LIN {X 0,Y 474.185,Z 288.904,A -85,B 0,C 180,E1 -7449.626,E2 -7449.626} C_VEL
LIN {X 0,Y 468.545,Z 295.09,A -85,B 0,C 180,E1 -7449.509,E2 -7449.509} C_VEL
LIN {X 0,Y 466.901,Z 298.538,A -85,B 0,C 180,E1 -7449.489,E2 -7449.489} C_VEL
LIN {X 0,Y 466.86,Z 301.446,A -85,B 0,C 180,E1 -7449.52,E2 -7449.52} C_VEL
LIN {X 0,Y 468.004,Z 304.741,A -85,B 0,C 180,E1 -7449.617,E2 -7449.617} C_VEL
LIN {X 0,Y 472.692,Z 312.938,A -85,B 0,C 180,E1 -7449.976,E2 -7449.976} C_VEL
LIN {X 0,Y 473.425,Z 316.419,A -85,B 0,C 180,E1 -7450.068,E2 -7450.068} C_VEL
LIN {X 0,Y 472.347,Z 423.939,A -85,B 0,C 180,E1 -7451.737,E2 -7451.737} C_VEL
LIN {X 0,Y 471.944,Z 437.997,A -85,B 0,C 180,E1 -7452.116,E2 -7452.116} C_VEL
LIN {X 0,Y 471.535,Z 451.556,A -85,B 0,C 180,E1 -7452.657,E2 -7452.657} C_VEL
LIN {X 0,Y 470.962,Z 463.993,A -85,B 0,C 180,E1 -7453.311,E2 -7453.311} C_VEL
LIN {X 0,Y 470.322,Z 476.852,A -85,B 0,C 180,E1 -7454.175,E2 -7454.175} C_VEL
LIN {X 0,Y 469.63,Z 488.571,A -85,B 0,C 180,E1 -7455.151,E2 -7455.151} C_VEL
LIN {X 0,Y 468.872,Z 500.266,A -85,B 0,C 180,E1 -7456.345,E2 -7456.345} C_VEL
LIN {X 0,Y 468.289,Z 510.754,A -85,B 0,C 180,E1 -7457.657,E2 -7457.657} C_VEL
LIN {X 0,Y 467.805,Z 519.328,A -85,B 0,C 180,E1 -7458.957,E2 -7458.957} C_VEL
LIN {X 0,Y 467.34,Z 527.589,A -85,B 0,C 180,E1 -7460.478,E2 -7460.478} C_VEL
LIN {X 0,Y 467.082,Z 533.343,A -85,B 0,C 180,E1 -7461.782,E2 -7461.782} C_VEL
LIN {X 0,Y 466.874,Z 539.353,A -85,B 0,C 180,E1 -7463.475,E2 -7463.475} C_VEL
LIN {X 0,Y 466.775,Z 542.98,A -85,B 0,C 180,E1 -7464.817,E2 -7464.817} C_VEL
LIN {X 0,Y 466.692,Z 546.396,A -85,B 0,C 180,E1 -7466.547,E2 -7466.547} C_VEL
LIN {X 0,Y 466.606,Z 548.426,A -85,B 0,C 180,E1 -7468.274,E2 -7468.274} C_VEL
LIN {X 0,Y 466.598,Z 549.126,A -85,B 0,C 180,E1 -7470,E2 -7470} C_VEL
LIN {X 0,Y 466.605,Z 548.504,A -85,B 0,C 180,E1 -7471.726,E2 -7471.726} C_VEL
LIN {X 0,Y 466.692,Z 546.544,A -85,B 0,C 180,E1 -7473.453,E2 -7473.453} C_VEL
LIN {X 0,Y 466.775,Z 543.2,A -85,B 0,C 180,E1 -7475.183,E2 -7475.183} C_VEL
LIN {X 0,Y 466.908,Z 538.376,A -85,B 0,C 180,E1 -7476.916,E2 -7476.916} C_VEL
LIN {X 0,Y 467.143,Z 531.917,A -85,B 0,C 180,E1 -7478.653,E2 -7478.653} C_VEL
LIN {X 0,Y 467.481,Z 524.725,A -85,B 0,C 180,E1 -7480.174,E2 -7480.174} C_VEL
LIN {X 0,Y 468.029,Z 515.83,A -85,B 0,C 180,E1 -7481.696,E2 -7481.696} C_VEL
LIN {X 0,Y 468.534,Z 506.485,A -85,B 0,C 180,E1 -7483.003,E2 -7483.003} C_VEL
LIN {X 0,Y 469.149,Z 496.136,A -85,B 0,C 180,E1 -7484.199,E2 -7484.199} C_VEL
LIN {X 0,Y 469.823,Z 484.715,A -85,B 0,C 180,E1 -7485.286,E2 -7485.286} C_VEL
LIN {X 0,Y 470.575,Z 472.057,A -85,B 0,C 180,E1 -7486.262,E2 -7486.262} C_VEL
LIN {X 0,Y 471.222,Z 458.762,A -85,B 0,C 180,E1 -7487.075,E2 -7487.075} C_VEL
LIN {X 0,Y 471.78,Z 444.827,A -85,B 0,C 180,E1 -7487.724,E2 -7487.724} C_VEL
LIN {X 0,Y 472.174,Z 431.019,A -85,B 0,C 180,E1 -7488.186,E2 -7488.186} C_VEL
LIN {X 0,Y 472.481,Z 416.795,A -85,B 0,C 180,E1 -7488.482,E2 -7488.482} C_VEL
LIN {X 0,Y 473.516,Z 306.855,A -85,B 0,C 180,E1 -7490.171,E2 -7490.171} C_VEL
LIN {X 0,Y 469.764,Z 287.63,A -85,B 0,C 180,E1 -7490.662,E2 -7490.662} C_VEL
LIN {X 0,Y 469.727,Z 286.836,A -85,B 0,C 180,E1 -7490.734,E2 -7490.734} C_VEL
LIN {X 0,Y 470.355,Z 273.557,A -85,B 0,C 180,E1 -7493.092,E2 -7493.092} C_VEL
LIN {X 0,Y 468.135,Z 262.406,A -85,B 0,C 180,E1 -7495.281,E2 -7495.281} C_VEL
LIN {X 0,Y 467.627,Z 259.921,A -85,B 0,C 180,E1 -7495.838,E2 -7495.838} C_VEL
LIN {X 0,Y 467.576,Z 259.854,A -85,B 0,C 180,E1 -7498.749,E2 -7498.749} C_VEL
LIN {X 0,Y 467.582,Z 259.864,A -85,B 0,C 180,E1 -7501.739,E2 -7501.739} C_VEL
LIN {X 0,Y 467.565,Z 259.863,A -85,B 0,C 180,E1 -7504.832,E2 -7504.832} C_VEL
LIN {X 0,Y 467.563,Z 259.863,A -85,B 0,C 180,E1 -7508.044,E2 -7508.044} C_VEL
LIN {X 0,Y 467.579,Z 259.863,A -85,B 0,C 180,E1 -7511.277,E2 -7511.277} C_VEL
LIN {X 0,Y 467.563,Z 259.867,A -85,B 0,C 180,E1 -7513.822,E2 -7513.822} C_VEL
LIN {X 0,Y 467.552,Z 259.865,A -85,B 0,C 180,E1 -7516.255,E2 -7516.255} C_VEL
LIN {X 0,Y 467.579,Z 259.848,A -85,B 0,C 180,E1 -7518.722,E2 -7518.722} C_VEL
LIN {X 0,Y 467.569,Z 259.871,A -85,B 0,C 180,E1 -7521.406,E2 -7521.406} C_VEL
LIN {X 0,Y 467.557,Z 259.863,A -85,B 0,C 180,E1 -7524.26,E2 -7524.26} C_VEL
LIN {X 0,Y 467.576,Z 259.848,A -85,B 0,C 180,E1 -7527.32,E2 -7527.32} C_VEL
LIN {X 0,Y 467.572,Z 259.866,A -85,B 0,C 180,E1 -7530.665,E2 -7530.665} C_VEL
LIN {X 0,Y 467.609,Z 259.858,A -85,B 0,C 180,E1 -7533.199,E2 -7533.199} C_VEL
LIN {X 0,Y 467.585,Z 259.864,A -85,B 0,C 180,E1 -7536.468,E2 -7536.468} C_VEL
LIN {X 0,Y 467.614,Z 259.853,A -85,B 0,C 180,E1 -7539.777,E2 -7539.777} C_VEL
LIN {X 0,Y 467.601,Z 259.863,A -85,B 0,C 180,E1 -7542.506,E2 -7542.506} C_VEL
LIN {X 0,Y 467.598,Z 259.858,A -85,B 0,C 180,E1 -7545.196,E2 -7545.196} C_VEL
LIN {X 0,Y 467.648,Z 259.854,A -85,B 0,C 180,E1 -7547.854,E2 -7547.854} C_VEL
LIN {X 0,Y 467.673,Z 259.845,A -85,B 0,C 180,E1 -7551.357,E2 -7551.357} C_VEL
LIN {X 0,Y 467.738,Z 259.843,A -85,B 0,C 180,E1 -7553.962,E2 -7553.962} C_VEL
LIN {X 0,Y 467.851,Z 259.819,A -85,B 0,C 180,E1 -7557.417,E2 -7557.417} C_VEL
LIN {X 0,Y 467.873,Z 259.826,A -85,B 0,C 180,E1 -7560,E2 -7560} C_VEL
LIN {X 0,Y 467.851,Z 259.828,A -85,B 0,C 180,E1 -7562.583,E2 -7562.583} C_VEL
LIN {X 0,Y 467.735,Z 259.843,A -85,B 0,C 180,E1 -7566.037,E2 -7566.037} C_VEL
LIN {X 0,Y 467.673,Z 259.85,A -85,B 0,C 180,E1 -7568.643,E2 -7568.643} C_VEL
LIN {X 0,Y 467.646,Z 259.856,A -85,B 0,C 180,E1 -7572.146,E2 -7572.146} C_VEL
LIN {X 0,Y 467.63,Z 259.855,A -85,B 0,C 180,E1 -7575.695,E2 -7575.695} C_VEL
LIN {X 0,Y 467.608,Z 259.86,A -85,B 0,C 180,E1 -7578.765,E2 -7578.765} C_VEL
LIN {X 0,Y 467.572,Z 259.86,A -85,B 0,C 180,E1 -7581.269,E2 -7581.269} C_VEL
LIN {X 0,Y 467.565,Z 259.867,A -85,B 0,C 180,E1 -7583.944,E2 -7583.944} C_VEL
LIN {X 0,Y 467.608,Z 259.854,A -85,B 0,C 180,E1 -7586.801,E2 -7586.801} C_VEL
LIN {X 0,Y 467.58,Z 259.867,A -85,B 0,C 180,E1 -7589.736,E2 -7589.736} C_VEL
LIN {X 0,Y 467.577,Z 259.852,A -85,B 0,C 180,E1 -7592.759,E2 -7592.759} C_VEL
LIN {X 0,Y 467.55,Z 259.856,A -85,B 0,C 180,E1 -7595.89,E2 -7595.89} C_VEL
LIN {X 0,Y 467.576,Z 259.864,A -85,B 0,C 180,E1 -7599.145,E2 -7599.145} C_VEL
LIN {X 0,Y 467.581,Z 259.863,A -85,B 0,C 180,E1 -7602.568,E2 -7602.568} C_VEL
LIN {X 0,Y 467.566,Z 259.865,A -85,B 0,C 180,E1 -7605.054,E2 -7605.054} C_VEL
LIN {X 0,Y 467.62,Z 259.855,A -85,B 0,C 180,E1 -7607.445,E2 -7607.445} C_VEL
LIN {X 0,Y 467.611,Z 259.861,A -85,B 0,C 180,E1 -7610.859,E2 -7610.859} C_VEL
LIN {X 0,Y 467.557,Z 259.868,A -85,B 0,C 180,E1 -7614.262,E2 -7614.262} C_VEL
LIN {X 0,Y 467.58,Z 259.865,A -85,B 0,C 180,E1 -7617.322,E2 -7617.322} C_VEL
LIN {X 0,Y 467.568,Z 259.845,A -85,B 0,C 180,E1 -7620.668,E2 -7620.668} C_VEL
LIN {X 0,Y 467.696,Z 259.995,A -85,B 0,C 180,E1 -7623.093,E2 -7623.093} C_VEL
LIN {X 0,Y 470.359,Z 272.736,A -85,B 0,C 180,E1 -7625.544,E2 -7625.544} C_VEL
LIN {X 0,Y 470.614,Z 276.547,A -85,B 0,C 180,E1 -7626.222,E2 -7626.222} C_VEL
LIN {X 0,Y 469.607,Z 295.051,A -85,B 0,C 180,E1 -7629.338,E2 -7629.338} C_VEL
LIN {X 0,Y 470.566,Z 300.147,A -85,B 0,C 180,E1 -7629.502,E2 -7629.502} C_VEL
LIN {X 0,Y 473.425,Z 315.558,A -85,B 0,C 180,E1 -7629.875,E2 -7629.875} C_VEL
LIN {X 0,Y 472.421,Z 422.331,A -85,B 0,C 180,E1 -7631.515,E2 -7631.515} C_VEL
LIN {X 0,Y 472.13,Z 437.826,A -85,B 0,C 180,E1 -7631.815,E2 -7631.815} C_VEL
LIN {X 0,Y 471.708,Z 451.895,A -85,B 0,C 180,E1 -7632.261,E2 -7632.261} C_VEL
LIN {X 0,Y 471.169,Z 465.576,A -85,B 0,C 180,E1 -7632.876,E2 -7632.876} C_VEL
LIN {X 0,Y 470.561,Z 478.308,A -85,B 0,C 180,E1 -7633.626,E2 -7633.626} C_VEL
LIN {X 0,Y 469.786,Z 491.398,A -85,B 0,C 180,E1 -7634.601,E2 -7634.601} C_VEL
LIN {X 0,Y 469.087,Z 503.159,A -85,B 0,C 180,E1 -7635.688,E2 -7635.688} C_VEL
LIN {X 0,Y 468.519,Z 512.899,A -85,B 0,C 180,E1 -7636.776,E2 -7636.776} C_VEL
LIN {X 0,Y 468.018,Z 522.641,A -85,B 0,C 180,E1 -7638.084,E2 -7638.084} C_VEL
LIN {X 0,Y 467.519,Z 530.722,A -85,B 0,C 180,E1 -7639.389,E2 -7639.389} C_VEL
LIN {X 0,Y 467.156,Z 538.466,A -85,B 0,C 180,E1 -7640.911,E2 -7640.911} C_VEL
LIN {X 0,Y 466.912,Z 543.872,A -85,B 0,C 180,E1 -7642.215,E2 -7642.215} C_VEL
LIN {X 0,Y 466.751,Z 549.559,A -85,B 0,C 180,E1 -7643.95,E2 -7643.95} C_VEL
LIN {X 0,Y 466.759,Z 551.808,A -85,B 0,C 180,E1 -7644.817,E2 -7644.817} C_VEL
LIN {X 0,Y 466.651,Z 555.204,A -85,B 0,C 180,E1 -7646.546,E2 -7646.546} C_VEL
LIN {X 0,Y 466.601,Z 557.214,A -85,B 0,C 180,E1 -7648.274,E2 -7648.274} C_VEL
LIN {X 0,Y 466.597,Z 557.88,A -85,B 0,C 180,E1 -7650,E2 -7650} C_VEL
LIN {X 0,Y 466.601,Z 557.214,A -85,B 0,C 180,E1 -7651.726,E2 -7651.726} C_VEL
LIN {X 0,Y 466.651,Z 555.207,A -85,B 0,C 180,E1 -7653.454,E2 -7653.454} C_VEL
LIN {X 0,Y 466.762,Z 551.809,A -85,B 0,C 180,E1 -7655.183,E2 -7655.183} C_VEL
LIN {X 0,Y 466.823,Z 546.916,A -85,B 0,C 180,E1 -7656.917,E2 -7656.917} C_VEL
LIN {X 0,Y 467.076,Z 540.386,A -85,B 0,C 180,E1 -7658.654,E2 -7658.654} C_VEL
LIN {X 0,Y 467.381,Z 533.119,A -85,B 0,C 180,E1 -7660.177,E2 -7660.177} C_VEL
LIN {X 0,Y 467.956,Z 524.12,A -85,B 0,C 180,E1 -7661.698,E2 -7661.698} C_VEL
LIN {X 0,Y 468.449,Z 514.673,A -85,B 0,C 180,E1 -7663.005,E2 -7663.005} C_VEL
LIN {X 0,Y 469.037,Z 504.214,A -85,B 0,C 180,E1 -7664.203,E2 -7664.203} C_VEL
LIN {X 0,Y 469.703,Z 492.673,A -85,B 0,C 180,E1 -7665.29,E2 -7665.29} C_VEL
LIN {X 0,Y 470.487,Z 479.869,A -85,B 0,C 180,E1 -7666.265,E2 -7666.265} C_VEL
LIN {X 0,Y 471.054,Z 468.255,A -85,B 0,C 180,E1 -7666.975,E2 -7666.975} C_VEL
LIN {X 0,Y 471.644,Z 454.226,A -85,B 0,C 180,E1 -7667.64,E2 -7667.64} C_VEL
LIN {X 0,Y 472.099,Z 439.998,A -85,B 0,C 180,E1 -7668.124,E2 -7668.124} C_VEL
LIN {X 0,Y 472.384,Z 425.772,A -85,B 0,C 180,E1 -7668.43,E2 -7668.43} C_VEL
LIN {X 0,Y 473.455,Z 315.776,A -85,B 0,C 180,E1 -7670.118,E2 -7670.118} C_VEL
LIN {X 0,Y 469.611,Z 295.324,A -85,B 0,C 180,E1 -7670.636,E2 -7670.636} C_VEL
LIN {X 0,Y 470.379,Z 280.548,A -85,B 0,C 180,E1 -7673.091,E2 -7673.091} C_VEL
LIN {X 0,Y 470.586,Z 274.299,A -85,B 0,C 180,E1 -7674.167,E2 -7674.167} C_VEL
LIN {X 0,Y 468.021,Z 261.697,A -85,B 0,C 180,E1 -7676.534,E2 -7676.534} C_VEL
LIN {X 0,Y 467.689,Z 259.904,A -85,B 0,C 180,E1 -7676.935,E2 -7676.935} C_VEL
LIN {X 0,Y 467.552,Z 259.845,A -85,B 0,C 180,E1 -7679.738,E2 -7679.738} C_VEL
LIN {X 0,Y 467.581,Z 259.863,A -85,B 0,C 180,E1 -7682.758,E2 -7682.758} C_VEL
LIN {X 0,Y 467.551,Z 259.869,A -85,B 0,C 180,E1 -7685.889,E2 -7685.889} C_VEL
LIN {X 0,Y 467.579,Z 259.865,A -85,B 0,C 180,E1 -7689.144,E2 -7689.144} C_VEL
LIN {X 0,Y 467.586,Z 259.86,A -85,B 0,C 180,E1 -7692.567,E2 -7692.567} C_VEL
LIN {X 0,Y 467.566,Z 259.864,A -85,B 0,C 180,E1 -7695.053,E2 -7695.053} C_VEL
LIN {X 0,Y 467.584,Z 259.863,A -85,B 0,C 180,E1 -7697.439,E2 -7697.439} C_VEL
LIN {X 0,Y 467.577,Z 259.864,A -85,B 0,C 180,E1 -7700.855,E2 -7700.855} C_VEL
LIN {X 0,Y 467.557,Z 259.852,A -85,B 0,C 180,E1 -7704.26,E2 -7704.26} C_VEL
LIN {X 0,Y 467.576,Z 259.853,A -85,B 0,C 180,E1 -7707.32,E2 -7707.32} C_VEL
LIN {X 0,Y 467.571,Z 259.864,A -85,B 0,C 180,E1 -7710.665,E2 -7710.665} C_VEL
LIN {X 0,Y 467.62,Z 259.853,A -85,B 0,C 180,E1 -7713.2,E2 -7713.2} C_VEL
LIN {X 0,Y 467.586,Z 259.86,A -85,B 0,C 180,E1 -7716.468,E2 -7716.468} C_VEL
LIN {X 0,Y 467.615,Z 259.862,A -85,B 0,C 180,E1 -7719.777,E2 -7719.777} C_VEL
LIN {X 0,Y 467.601,Z 259.855,A -85,B 0,C 180,E1 -7722.507,E2 -7722.507} C_VEL
LIN {X 0,Y 467.598,Z 259.859,A -85,B 0,C 180,E1 -7725.196,E2 -7725.196} C_VEL
LIN {X 0,Y 467.647,Z 259.856,A -85,B 0,C 180,E1 -7727.854,E2 -7727.854} C_VEL
LIN {X 0,Y 467.674,Z 259.85,A -85,B 0,C 180,E1 -7731.357,E2 -7731.357} C_VEL
LIN {X 0,Y 467.735,Z 259.843,A -85,B 0,C 180,E1 -7733.963,E2 -7733.963} C_VEL
LIN {X 0,Y 467.852,Z 259.828,A -85,B 0,C 180,E1 -7737.417,E2 -7737.417} C_VEL
LIN {X 0,Y 467.874,Z 259.826,A -85,B 0,C 180,E1 -7740,E2 -7740} C_VEL
LIN {X 0,Y 467.852,Z 259.818,A -85,B 0,C 180,E1 -7742.583,E2 -7742.583} C_VEL
LIN {X 0,Y 467.739,Z 259.843,A -85,B 0,C 180,E1 -7746.038,E2 -7746.038} C_VEL
LIN {X 0,Y 467.674,Z 259.844,A -85,B 0,C 180,E1 -7748.643,E2 -7748.643} C_VEL
LIN {X 0,Y 467.648,Z 259.854,A -85,B 0,C 180,E1 -7752.146,E2 -7752.146} C_VEL
LIN {X 0,Y 467.631,Z 259.855,A -85,B 0,C 180,E1 -7755.695,E2 -7755.695} C_VEL
LIN {X 0,Y 467.61,Z 259.862,A -85,B 0,C 180,E1 -7758.765,E2 -7758.765} C_VEL
LIN {X 0,Y 467.573,Z 259.863,A -85,B 0,C 180,E1 -7761.269,E2 -7761.269} C_VEL
LIN {X 0,Y 467.566,Z 259.864,A -85,B 0,C 180,E1 -7763.944,E2 -7763.944} C_VEL
LIN {X 0,Y 467.61,Z 259.857,A -85,B 0,C 180,E1 -7766.801,E2 -7766.801} C_VEL
LIN {X 0,Y 467.581,Z 259.861,A -85,B 0,C 180,E1 -7769.736,E2 -7769.736} C_VEL
LIN {X 0,Y 467.578,Z 259.846,A -85,B 0,C 180,E1 -7772.759,E2 -7772.759} C_VEL
LIN {X 0,Y 467.552,Z 259.861,A -85,B 0,C 180,E1 -7775.89,E2 -7775.89} C_VEL
LIN {X 0,Y 467.593,Z 259.859,A -85,B 0,C 180,E1 -7779.144,E2 -7779.144} C_VEL
LIN {X 0,Y 467.582,Z 259.852,A -85,B 0,C 180,E1 -7782.568,E2 -7782.568} C_VEL
LIN {X 0,Y 467.567,Z 259.867,A -85,B 0,C 180,E1 -7785.054,E2 -7785.054} C_VEL
LIN {X 0,Y 467.586,Z 259.85,A -85,B 0,C 180,E1 -7787.441,E2 -7787.441} C_VEL
LIN {X 0,Y 467.58,Z 259.864,A -85,B 0,C 180,E1 -7790.856,E2 -7790.856} C_VEL
LIN {X 0,Y 467.561,Z 259.87,A -85,B 0,C 180,E1 -7794.261,E2 -7794.261} C_VEL
LIN {X 0,Y 467.581,Z 259.865,A -85,B 0,C 180,E1 -7797.322,E2 -7797.322} C_VEL
LIN {X 0,Y 467.57,Z 259.862,A -85,B 0,C 180,E1 -7800.668,E2 -7800.668} C_VEL
LIN {X 0,Y 467.614,Z 259.859,A -85,B 0,C 180,E1 -7803.2,E2 -7803.2} C_VEL
LIN {X 0,Y 467.651,Z 260.072,A -85,B 0,C 180,E1 -7804.322,E2 -7804.322} C_VEL
LIN {X 0,Y 470.316,Z 273.054,A -85,B 0,C 180,E1 -7806.905,E2 -7806.905} C_VEL
LIN {X 0,Y 469.832,Z 284.512,A -85,B 0,C 180,E1 -7808.961,E2 -7808.961} C_VEL
LIN {X 0,Y 469.725,Z 287.474,A -85,B 0,C 180,E1 -7809.425,E2 -7809.425} C_VEL
LIN {X 0,Y 473.448,Z 305.821,A -85,B 0,C 180,E1 -7809.902,E2 -7809.902} C_VEL
LIN {X 0,Y 473.425,Z 316.419,A -85,B 0,C 180,E1 -7810.068,E2 -7810.068} C_VEL
LIN {X 0,Y 472.794,Z 322.27,A -85,B 0,C 180,E1 -7810.133,E2 -7810.133} C_VEL
LIN {X 0,Y 467.131,Z 341.305,A -85,B 0,C 180,E1 -7810.186,E2 -7810.186} C_VEL
LIN {X 0,Y 466.478,Z 347.157,A -85,B 0,C 180,E1 -7810.251,E2 -7810.251} C_VEL
LIN {X 0,Y 465.631,Z 424.025,A -85,B 0,C 180,E1 -7811.464,E2 -7811.464} C_VEL
LIN {X 0,Y 465.192,Z 438.076,A -85,B 0,C 180,E1 -7811.848,E2 -7811.848} C_VEL
LIN {X 0,Y 464.766,Z 451.632,A -85,B 0,C 180,E1 -7812.397,E2 -7812.397} C_VEL
LIN {X 0,Y 464.164,Z 464.224,A -85,B 0,C 180,E1 -7813.069,E2 -7813.069} C_VEL
LIN {X 0,Y 463.481,Z 476.925,A -85,B 0,C 180,E1 -7813.935,E2 -7813.935} C_VEL
LIN {X 0,Y 462.728,Z 488.643,A -85,B 0,C 180,E1 -7814.924,E2 -7814.924} C_VEL
LIN {X 0,Y 461.946,Z 500.337,A -85,B 0,C 180,E1 -7816.136,E2 -7816.136} C_VEL
LIN {X 0,Y 461.318,Z 509.8,A -85,B 0,C 180,E1 -7817.326,E2 -7817.326} C_VEL
LIN {X 0,Y 460.916,Z 518.046,A -85,B 0,C 180,E1 -7818.567,E2 -7818.567} C_VEL
LIN {X 0,Y 460.472,Z 525.443,A -85,B 0,C 180,E1 -7819.891,E2 -7819.891} C_VEL
LIN {X 0,Y 460.11,Z 531.608,A -85,B 0,C 180,E1 -7821.214,E2 -7821.214} C_VEL
LIN {X 0,Y 459.839,Z 538.145,A -85,B 0,C 180,E1 -7822.977,E2 -7822.977} C_VEL
LIN {X 0,Y 459.712,Z 543.048,A -85,B 0,C 180,E1 -7824.737,E2 -7824.737} C_VEL
LIN {X 0,Y 459.59,Z 546.463,A -85,B 0,C 180,E1 -7826.493,E2 -7826.493} C_VEL
LIN {X 0,Y 459.519,Z 548.493,A -85,B 0,C 180,E1 -7828.247,E2 -7828.247} C_VEL
LIN {X 0,Y 459.5,Z 549.193,A -85,B 0,C 180,E1 -7830,E2 -7830} C_VEL
LIN {X 0,Y 459.518,Z 548.57,A -85,B 0,C 180,E1 -7831.753,E2 -7831.753} C_VEL
LIN {X 0,Y 459.589,Z 546.61,A -85,B 0,C 180,E1 -7833.507,E2 -7833.507} C_VEL
LIN {X 0,Y 459.712,Z 543.266,A -85,B 0,C 180,E1 -7835.263,E2 -7835.263} C_VEL
LIN {X 0,Y 459.842,Z 538.441,A -85,B 0,C 180,E1 -7837.023,E2 -7837.023} C_VEL
LIN {X 0,Y 460.094,Z 531.982,A -85,B 0,C 180,E1 -7838.786,E2 -7838.786} C_VEL
LIN {X 0,Y 460.458,Z 524.789,A -85,B 0,C 180,E1 -7840.331,E2 -7840.331} C_VEL
LIN {X 0,Y 461.05,Z 515.894,A -85,B 0,C 180,E1 -7841.875,E2 -7841.875} C_VEL
LIN {X 0,Y 461.588,Z 506.549,A -85,B 0,C 180,E1 -7843.202,E2 -7843.202} C_VEL
LIN {X 0,Y 462.228,Z 496.198,A -85,B 0,C 180,E1 -7844.417,E2 -7844.417} C_VEL
LIN {X 0,Y 462.965,Z 484.777,A -85,B 0,C 180,E1 -7845.518,E2 -7845.518} C_VEL
LIN {X 0,Y 463.757,Z 472.118,A -85,B 0,C 180,E1 -7846.507,E2 -7846.507} C_VEL
LIN {X 0,Y 464.416,Z 459.403,A -85,B 0,C 180,E1 -7847.299,E2 -7847.299} C_VEL
LIN {X 0,Y 464.971,Z 446.183,A -85,B 0,C 180,E1 -7847.936,E2 -7847.936} C_VEL
LIN {X 0,Y 465.385,Z 432.904,A -85,B 0,C 180,E1 -7848.403,E2 -7848.403} C_VEL
LIN {X 0,Y 465.7,Z 418.442,A -85,B 0,C 180,E1 -7848.733,E2 -7848.733} C_VEL
LIN {X 0,Y 466.859,Z 307.527,A -85,B 0,C 180,E1 -7850.462,E2 -7850.462} C_VEL
LIN {X 0,Y 462.855,Z 287.376,A -85,B 0,C 180,E1 -7851,E2 -7851} C_VEL
LIN {X 0,Y 463.435,Z 274.89,A -85,B 0,C 180,E1 -7853.221,E2 -7853.221} C_VEL
LIN {X 0,Y 460.776,Z 261.727,A -85,B 0,C 180,E1 -7855.855,E2 -7855.855} C_VEL
LIN {X 0,Y 460.571,Z 260.769,A -85,B 0,C 180,E1 -7856.129,E2 -7856.129} C_VEL
LIN {X 0,Y 460.539,Z 260.735,A -85,B 0,C 180,E1 -7859.23,E2 -7859.23} C_VEL
LIN {X 0,Y 460.53,Z 260.744,A -85,B 0,C 180,E1 -7862.284,E2 -7862.284} C_VEL
LIN {X 0,Y 460.511,Z 260.748,A -85,B 0,C 180,E1 -7865.445,E2 -7865.445} C_VEL
LIN {X 0,Y 460.542,Z 260.738,A -85,B 0,C 180,E1 -7868.897,E2 -7868.897} C_VEL
LIN {X 0,Y 460.52,Z 260.731,A -85,B 0,C 180,E1 -7872.18,E2 -7872.18} C_VEL
LIN {X 0,Y 460.513,Z 260.749,A -85,B 0,C 180,E1 -7875.411,E2 -7875.411} C_VEL
LIN {X 0,Y 460.531,Z 260.725,A -85,B 0,C 180,E1 -7878.396,E2 -7878.396} C_VEL
LIN {X 0,Y 460.539,Z 260.744,A -85,B 0,C 180,E1 -7881.268,E2 -7881.268} C_VEL
LIN {X 0,Y 460.508,Z 260.742,A -85,B 0,C 180,E1 -7884.554,E2 -7884.554} C_VEL
LIN {X 0,Y 460.526,Z 260.73,A -85,B 0,C 180,E1 -7887.715,E2 -7887.715} C_VEL
LIN {X 0,Y 460.541,Z 260.743,A -85,B 0,C 180,E1 -7890.769,E2 -7890.769} C_VEL
LIN {X 0,Y 460.555,Z 260.732,A -85,B 0,C 180,E1 -7893.734,E2 -7893.734} C_VEL
LIN {X 0,Y 460.538,Z 260.743,A -85,B 0,C 180,E1 -7896.623,E2 -7896.623} C_VEL
LIN {X 0,Y 460.543,Z 260.736,A -85,B 0,C 180,E1 -7899.452,E2 -7899.452} C_VEL
LIN {X 0,Y 460.551,Z 260.739,A -85,B 0,C 180,E1 -7902.23,E2 -7902.23} C_VEL
LIN {X 0,Y 460.557,Z 260.734,A -85,B 0,C 180,E1 -7904.964,E2 -7904.964} C_VEL
LIN {X 0,Y 460.605,Z 260.737,A -85,B 0,C 180,E1 -7908.559,E2 -7908.559} C_VEL
LIN {X 0,Y 460.686,Z 260.715,A -85,B 0,C 180,E1 -7912.108,E2 -7912.108} C_VEL
LIN {X 0,Y 460.692,Z 260.726,A -85,B 0,C 180,E1 -7914.748,E2 -7914.748} C_VEL
LIN {X 0,Y 460.817,Z 260.695,A -85,B 0,C 180,E1 -7917.378,E2 -7917.378} C_VEL
LIN {X 0,Y 460.844,Z 260.702,A -85,B 0,C 180,E1 -7920,E2 -7920} C_VEL
LIN {X 0,Y 460.816,Z 260.704,A -85,B 0,C 180,E1 -7922.622,E2 -7922.622} C_VEL
LIN {X 0,Y 460.701,Z 260.72,A -85,B 0,C 180,E1 -7926.13,E2 -7926.13} C_VEL
LIN {X 0,Y 460.62,Z 260.727,A -85,B 0,C 180,E1 -7928.776,E2 -7928.776} C_VEL
LIN {X 0,Y 460.604,Z 260.738,A -85,B 0,C 180,E1 -7932.445,E2 -7932.445} C_VEL
LIN {X 0,Y 460.591,Z 260.732,A -85,B 0,C 180,E1 -7935.998,E2 -7935.998} C_VEL
LIN {X 0,Y 460.562,Z 260.737,A -85,B 0,C 180,E1 -7938.902,E2 -7938.902} C_VEL
LIN {X 0,Y 460.508,Z 260.741,A -85,B 0,C 180,E1 -7941.486,E2 -7941.486} C_VEL
LIN {X 0,Y 460.535,Z 260.745,A -85,B 0,C 180,E1 -7944.333,E2 -7944.333} C_VEL
LIN {X 0,Y 460.571,Z 260.73,A -85,B 0,C 180,E1 -7947.244,E2 -7947.244} C_VEL
LIN {X 0,Y 460.52,Z 260.745,A -85,B 0,C 180,E1 -7950.239,E2 -7950.239} C_VEL
LIN {X 0,Y 460.522,Z 260.731,A -85,B 0,C 180,E1 -7953.325,E2 -7953.325} C_VEL
LIN {X 0,Y 460.472,Z 260.745,A -85,B 0,C 180,E1 -7956.53,E2 -7956.53} C_VEL
LIN {X 0,Y 460.552,Z 260.74,A -85,B 0,C 180,E1 -7959.86,E2 -7959.86} C_VEL
LIN {X 0,Y 460.508,Z 260.744,A -85,B 0,C 180,E1 -7962.901,E2 -7962.901} C_VEL
LIN {X 0,Y 460.519,Z 260.747,A -85,B 0,C 180,E1 -7965.829,E2 -7965.829} C_VEL
LIN {X 0,Y 460.539,Z 260.73,A -85,B 0,C 180,E1 -7968.991,E2 -7968.991} C_VEL
LIN {X 0,Y 460.54,Z 260.745,A -85,B 0,C 180,E1 -7971.269,E2 -7971.269} C_VEL
LIN {X 0,Y 460.507,Z 260.746,A -85,B 0,C 180,E1 -7974.555,E2 -7974.555} C_VEL
LIN {X 0,Y 460.529,Z 260.747,A -85,B 0,C 180,E1 -7977.716,E2 -7977.716} C_VEL
LIN {X 0,Y 460.538,Z 260.72,A -85,B 0,C 180,E1 -7980.77,E2 -7980.77} C_VEL
LIN {X 0,Y 460.668,Z 260.876,A -85,B 0,C 180,E1 -7982.824,E2 -7982.824} C_VEL
LIN {X 0,Y 463.302,Z 273.424,A -85,B 0,C 180,E1 -7985.279,E2 -7985.279} C_VEL
LIN {X 0,Y 463.746,Z 277.829,A -85,B 0,C 180,E1 -7986.085,E2 -7986.085} C_VEL
LIN {X 0,Y 462.744,Z 295.197,A -85,B 0,C 180,E1 -7989.036,E2 -7989.036} C_VEL
LIN {X 0,Y 466.7,Z 316.081,A -85,B 0,C 180,E1 -7989.582,E2 -7989.582} C_VEL
LIN {X 0,Y 465.883,Z 407.969,A -85,B 0,C 180,E1 -7991.018,E2 -7991.018} C_VEL
LIN {X 0,Y 465.535,Z 434.234,A -85,B 0,C 180,E1 -7991.46,E2 -7991.46} C_VEL
LIN {X 0,Y 465.024,Z 448.343,A -85,B 0,C 180,E1 -7991.867,E2 -7991.867} C_VEL
LIN {X 0,Y 464.517,Z 461.96,A -85,B 0,C 180,E1 -7992.441,E2 -7992.441} C_VEL
LIN {X 0,Y 463.879,Z 475.149,A -85,B 0,C 180,E1 -7993.178,E2 -7993.178} C_VEL
LIN {X 0,Y 463.207,Z 487.295,A -85,B 0,C 180,E1 -7994.038,E2 -7994.038} C_VEL
LIN {X 0,Y 462.469,Z 498.686,A -85,B 0,C 180,E1 -7995.029,E2 -7995.029} C_VEL
LIN {X 0,Y 461.799,Z 509.154,A -85,B 0,C 180,E1 -7996.132,E2 -7996.132} C_VEL
LIN {X 0,Y 461.214,Z 519.016,A -85,B 0,C 180,E1 -7997.383,E2 -7997.383} C_VEL
LIN {X 0,Y 460.699,Z 528.157,A -85,B 0,C 180,E1 -7998.785,E2 -7998.785} C_VEL
LIN {X 0,Y 460.224,Z 536.382,A -85,B 0,C 180,E1 -8000.33,E2 -8000.33} C_VEL
LIN {X 0,Y 459.931,Z 542.138,A -85,B 0,C 180,E1 -8001.653,E2 -8001.653} C_VEL
LIN {X 0,Y 459.739,Z 546.855,A -85,B 0,C 180,E1 -8002.976,E2 -8002.976} C_VEL
LIN {X 0,Y 459.669,Z 551.741,A -85,B 0,C 180,E1 -8004.737,E2 -8004.737} C_VEL
LIN {X 0,Y 459.548,Z 555.138,A -85,B 0,C 180,E1 -8006.493,E2 -8006.493} C_VEL
LIN {X 0,Y 459.514,Z 557.147,A -85,B 0,C 180,E1 -8008.247,E2 -8008.247} C_VEL
LIN {X 0,Y 459.499,Z 557.813,A -85,B 0,C 180,E1 -8010,E2 -8010} C_VEL
LIN {X 0,Y 459.514,Z 557.148,A -85,B 0,C 180,E1 -8011.753,E2 -8011.753} C_VEL
LIN {X 0,Y 459.548,Z 555.14,A -85,B 0,C 180,E1 -8013.507,E2 -8013.507} C_VEL
LIN {X 0,Y 459.673,Z 551.742,A -85,B 0,C 180,E1 -8015.263,E2 -8015.263} C_VEL
LIN {X 0,Y 459.734,Z 546.848,A -85,B 0,C 180,E1 -8017.025,E2 -8017.025} C_VEL
LIN {X 0,Y 460.022,Z 540.318,A -85,B 0,C 180,E1 -8018.788,E2 -8018.788} C_VEL
LIN {X 0,Y 460.353,Z 533.051,A -85,B 0,C 180,E1 -8020.334,E2 -8020.334} C_VEL
LIN {X 0,Y 460.962,Z 524.051,A -85,B 0,C 180,E1 -8021.878,E2 -8021.878} C_VEL
LIN {X 0,Y 461.501,Z 514.604,A -85,B 0,C 180,E1 -8023.204,E2 -8023.204} C_VEL
LIN {X 0,Y 462.135,Z 504.145,A -85,B 0,C 180,E1 -8024.42,E2 -8024.42} C_VEL
LIN {X 0,Y 462.829,Z 492.603,A -85,B 0,C 180,E1 -8025.523,E2 -8025.523} C_VEL
LIN {X 0,Y 463.644,Z 479.798,A -85,B 0,C 180,E1 -8026.512,E2 -8026.512} C_VEL
LIN {X 0,Y 464.321,Z 467.043,A -85,B 0,C 180,E1 -8027.294,E2 -8027.294} C_VEL
LIN {X 0,Y 464.869,Z 454.153,A -85,B 0,C 180,E1 -8027.906,E2 -8027.906} C_VEL
LIN {X 0,Y 465.36,Z 439.923,A -85,B 0,C 180,E1 -8028.396,E2 -8028.396} C_VEL
LIN {X 0,Y 465.676,Z 425.69,A -85,B 0,C 180,E1 -8028.705,E2 -8028.705} C_VEL
LIN {X 0,Y 466.796,Z 316.746,A -85,B 0,C 180,E1 -8030.4,E2 -8030.4} C_VEL
LIN {X 0,Y 462.732,Z 295.266,A -85,B 0,C 180,E1 -8030.956,E2 -8030.956} C_VEL
LIN {X 0,Y 463.286,Z 284.511,A -85,B 0,C 180,E1 -8032.757,E2 -8032.757} C_VEL
LIN {X 0,Y 463.727,Z 276.456,A -85,B 0,C 180,E1 -8034.154,E2 -8034.154} C_VEL
LIN {X 0,Y 461.671,Z 265.683,A -85,B 0,C 180,E1 -8036.197,E2 -8036.197} C_VEL
LIN {X 0,Y 460.668,Z 260.851,A -85,B 0,C 180,E1 -8037.176,E2 -8037.176} C_VEL
LIN {X 0,Y 460.509,Z 260.724,A -85,B 0,C 180,E1 -8040.239,E2 -8040.239} C_VEL
LIN {X 0,Y 460.527,Z 260.737,A -85,B 0,C 180,E1 -8043.324,E2 -8043.324} C_VEL
LIN {X 0,Y 460.473,Z 260.745,A -85,B 0,C 180,E1 -8046.529,E2 -8046.529} C_VEL
LIN {X 0,Y 460.529,Z 260.744,A -85,B 0,C 180,E1 -8049.862,E2 -8049.862} C_VEL
LIN {X 0,Y 460.516,Z 260.743,A -85,B 0,C 180,E1 -8052.901,E2 -8052.901} C_VEL
LIN {X 0,Y 460.507,Z 260.745,A -85,B 0,C 180,E1 -8055.83,E2 -8055.83} C_VEL
LIN {X 0,Y 460.526,Z 260.738,A -85,B 0,C 180,E1 -8058.988,E2 -8058.988} C_VEL
LIN {X 0,Y 460.521,Z 260.742,A -85,B 0,C 180,E1 -8061.266,E2 -8061.266} C_VEL
LIN {X 0,Y 460.508,Z 260.725,A -85,B 0,C 180,E1 -8064.554,E2 -8064.554} C_VEL
LIN {X 0,Y 460.526,Z 260.734,A -85,B 0,C 180,E1 -8067.715,E2 -8067.715} C_VEL
LIN {X 0,Y 460.541,Z 260.739,A -85,B 0,C 180,E1 -8070.769,E2 -8070.769} C_VEL
LIN {X 0,Y 460.561,Z 260.736,A -85,B 0,C 180,E1 -8073.735,E2 -8073.735} C_VEL
LIN {X 0,Y 460.539,Z 260.736,A -85,B 0,C 180,E1 -8076.624,E2 -8076.624} C_VEL
LIN {X 0,Y 460.543,Z 260.739,A -85,B 0,C 180,E1 -8079.452,E2 -8079.452} C_VEL
LIN {X 0,Y 460.551,Z 260.735,A -85,B 0,C 180,E1 -8082.23,E2 -8082.23} C_VEL
LIN {X 0,Y 460.557,Z 260.734,A -85,B 0,C 180,E1 -8084.965,E2 -8084.965} C_VEL
LIN {X 0,Y 460.603,Z 260.727,A -85,B 0,C 180,E1 -8088.559,E2 -8088.559} C_VEL
LIN {X 0,Y 460.687,Z 260.723,A -85,B 0,C 180,E1 -8092.108,E2 -8092.108} C_VEL
LIN {X 0,Y 460.69,Z 260.717,A -85,B 0,C 180,E1 -8094.748,E2 -8094.748} C_VEL
LIN {X 0,Y 460.817,Z 260.703,A -85,B 0,C 180,E1 -8097.378,E2 -8097.378} C_VEL
LIN {X 0,Y 460.844,Z 260.702,A -85,B 0,C 180,E1 -8100,E2 -8100} C_VEL
LIN {X 0,Y 460.817,Z 260.694,A -85,B 0,C 180,E1 -8102.622,E2 -8102.622} C_VEL
LIN {X 0,Y 460.705,Z 260.719,A -85,B 0,C 180,E1 -8106.13,E2 -8106.13} C_VEL
LIN {X 0,Y 460.621,Z 260.723,A -85,B 0,C 180,E1 -8108.776,E2 -8108.776} C_VEL
LIN {X 0,Y 460.605,Z 260.731,A -85,B 0,C 180,E1 -8112.445,E2 -8112.445} C_VEL
LIN {X 0,Y 460.592,Z 260.73,A -85,B 0,C 180,E1 -8115.998,E2 -8115.998} C_VEL
LIN {X 0,Y 460.563,Z 260.741,A -85,B 0,C 180,E1 -8118.902,E2 -8118.902} C_VEL
LIN {X 0,Y 460.508,Z 260.744,A -85,B 0,C 180,E1 -8121.486,E2 -8121.486} C_VEL
LIN {X 0,Y 460.536,Z 260.741,A -85,B 0,C 180,E1 -8124.333,E2 -8124.333} C_VEL
LIN {X 0,Y 460.573,Z 260.739,A -85,B 0,C 180,E1 -8127.244,E2 -8127.244} C_VEL
LIN {X 0,Y 460.522,Z 260.741,A -85,B 0,C 180,E1 -8130.239,E2 -8130.239} C_VEL
LIN {X 0,Y 460.524,Z 260.719,A -85,B 0,C 180,E1 -8133.325,E2 -8133.325} C_VEL
LIN {X 0,Y 460.474,Z 260.747,A -85,B 0,C 180,E1 -8136.53,E2 -8136.53} C_VEL
LIN {X 0,Y 460.568,Z 260.731,A -85,B 0,C 180,E1 -8139.859,E2 -8139.859} C_VEL
LIN {X 0,Y 460.51,Z 260.738,A -85,B 0,C 180,E1 -8142.901,E2 -8142.901} C_VEL
LIN {X 0,Y 460.516,Z 260.742,A -85,B 0,C 180,E1 -8145.83,E2 -8145.83} C_VEL
LIN {X 0,Y 460.531,Z 260.743,A -85,B 0,C 180,E1 -8148.99,E2 -8148.99} C_VEL
LIN {X 0,Y 460.524,Z 260.739,A -85,B 0,C 180,E1 -8151.268,E2 -8151.268} C_VEL
LIN {X 0,Y 460.511,Z 260.748,A -85,B 0,C 180,E1 -8154.555,E2 -8154.555} C_VEL
LIN {X 0,Y 460.531,Z 260.744,A -85,B 0,C 180,E1 -8157.716,E2 -8157.716} C_VEL
LIN {X 0,Y 460.539,Z 260.736,A -85,B 0,C 180,E1 -8160.77,E2 -8160.77} C_VEL
LIN {X 0,Y 460.559,Z 260.743,A -85,B 0,C 180,E1 -8163.735,E2 -8163.735} C_VEL
LIN {X 0,Y 460.608,Z 261.037,A -85,B 0,C 180,E1 -8164.082,E2 -8164.082} C_VEL
LIN {X 0,Y 463.363,Z 274.392,A -85,B 0,C 180,E1 -8166.775,E2 -8166.775} C_VEL
LIN {X 0,Y 463.176,Z 280.434,A -85,B 0,C 180,E1 -8167.883,E2 -8167.883} C_VEL
LIN {X 0,Y 462.838,Z 287.29,A -85,B 0,C 180,E1 -8169.086,E2 -8169.086} C_VEL
LIN {X 0,Y 465.8,Z 301.91,A -85,B 0,C 180,E1 -8169.492,E2 -8169.492} C_VEL
LIN {X 0,Y 466.834,Z 307.245,A -85,B 0,C 180,E1 -8169.626,E2 -8169.626} C_VEL
LIN {X 0,Y 466.478,Z 347.157,A -85,B 0,C 180,E1 -8170.251,E2 -8170.251} C_VEL
LIN {X 0,Y 465.841,Z 353.002,A -85,B 0,C 180,E1 -8170.316,E2 -8170.316} C_VEL
LIN {X 0,Y 460.227,Z 372.029,A -85,B 0,C 180,E1 -8170.374,E2 -8170.374} C_VEL
LIN {X 0,Y 459.538,Z 377.877,A -85,B 0,C 180,E1 -8170.438,E2 -8170.438} C_VEL
LIN {X 0,Y 458.916,Z 424.112,A -85,B 0,C 180,E1 -8171.183,E2 -8171.183} C_VEL
LIN {X 0,Y 458.477,Z 438.155,A -85,B 0,C 180,E1 -8171.572,E2 -8171.572} C_VEL
LIN {X 0,Y 457.996,Z 451.707,A -85,B 0,C 180,E1 -8172.128,E2 -8172.128} C_VEL
LIN {X 0,Y 457.366,Z 464.485,A -85,B 0,C 180,E1 -8172.822,E2 -8172.822} C_VEL
LIN {X 0,Y 456.627,Z 476.997,A -85,B 0,C 180,E1 -8173.687,E2 -8173.687} C_VEL
LIN {X 0,Y 455.827,Z 488.715,A -85,B 0,C 180,E1 -8174.691,E2 -8174.691} C_VEL
LIN {X 0,Y 455.04,Z 500.408,A -85,B 0,C 180,E1 -8175.921,E2 -8175.921} C_VEL
LIN {X 0,Y 454.324,Z 510.451,A -85,B 0,C 180,E1 -8177.209,E2 -8177.209} C_VEL
LIN {X 0,Y 453.838,Z 519.467,A -85,B 0,C 180,E1 -8178.613,E2 -8178.613} C_VEL
LIN {X 0,Y 453.321,Z 527.727,A -85,B 0,C 180,E1 -8180.181,E2 -8180.181} C_VEL
LIN {X 0,Y 452.98,Z 533.481,A -85,B 0,C 180,E1 -8181.524,E2 -8181.524} C_VEL
LIN {X 0,Y 452.754,Z 538.214,A -85,B 0,C 180,E1 -8182.867,E2 -8182.867} C_VEL
LIN {X 0,Y 452.627,Z 543.116,A -85,B 0,C 180,E1 -8184.654,E2 -8184.654} C_VEL
LIN {X 0,Y 452.489,Z 546.531,A -85,B 0,C 180,E1 -8186.438,E2 -8186.438} C_VEL
LIN {X 0,Y 452.435,Z 548.56,A -85,B 0,C 180,E1 -8188.22,E2 -8188.22} C_VEL
LIN {X 0,Y 452.406,Z 549.26,A -85,B 0,C 180,E1 -8190,E2 -8190} C_VEL
LIN {X 0,Y 452.435,Z 548.636,A -85,B 0,C 180,E1 -8191.78,E2 -8191.78} C_VEL
LIN {X 0,Y 452.488,Z 546.676,A -85,B 0,C 180,E1 -8193.562,E2 -8193.562} C_VEL
LIN {X 0,Y 452.628,Z 543.331,A -85,B 0,C 180,E1 -8195.345,E2 -8195.345} C_VEL
LIN {X 0,Y 452.755,Z 538.507,A -85,B 0,C 180,E1 -8197.133,E2 -8197.133} C_VEL
LIN {X 0,Y 453.062,Z 532.047,A -85,B 0,C 180,E1 -8198.924,E2 -8198.924} C_VEL
LIN {X 0,Y 453.424,Z 524.854,A -85,B 0,C 180,E1 -8200.493,E2 -8200.493} C_VEL
LIN {X 0,Y 454.072,Z 515.958,A -85,B 0,C 180,E1 -8202.06,E2 -8202.06} C_VEL
LIN {X 0,Y 454.65,Z 506.612,A -85,B 0,C 180,E1 -8203.407,E2 -8203.407} C_VEL
LIN {X 0,Y 455.341,Z 496.261,A -85,B 0,C 180,E1 -8204.639,E2 -8204.639} C_VEL
LIN {X 0,Y 456.098,Z 484.838,A -85,B 0,C 180,E1 -8205.758,E2 -8205.758} C_VEL
LIN {X 0,Y 456.937,Z 472.178,A -85,B 0,C 180,E1 -8206.761,E2 -8206.761} C_VEL
LIN {X 0,Y 457.676,Z 458.7,A -85,B 0,C 180,E1 -8207.607,E2 -8207.607} C_VEL
LIN {X 0,Y 458.251,Z 445.956,A -85,B 0,C 180,E1 -8208.221,E2 -8208.221} C_VEL
LIN {X 0,Y 458.676,Z 432.221,A -85,B 0,C 180,E1 -8208.706,E2 -8208.706} C_VEL
LIN {X 0,Y 459.003,Z 418.485,A -85,B 0,C 180,E1 -8209.016,E2 -8209.016} C_VEL
LIN {X 0,Y 460.164,Z 307.893,A -85,B 0,C 180,E1 -8210.768,E2 -8210.768} C_VEL
LIN {X 0,Y 455.996,Z 287.434,A -85,B 0,C 180,E1 -8211.331,E2 -8211.331} C_VEL
LIN {X 0,Y 456.52,Z 276.224,A -85,B 0,C 180,E1 -8213.354,E2 -8213.354} C_VEL
LIN {X 0,Y 453.78,Z 262.9,A -85,B 0,C 180,E1 -8216.066,E2 -8216.066} C_VEL
LIN {X 0,Y 453.522,Z 261.647,A -85,B 0,C 180,E1 -8216.414,E2 -8216.414} C_VEL
LIN {X 0,Y 453.509,Z 261.604,A -85,B 0,C 180,E1 -8218.711,E2 -8218.711} C_VEL
LIN {X 0,Y 453.463,Z 261.623,A -85,B 0,C 180,E1 -8221.799,E2 -8221.799} C_VEL
LIN {X 0,Y 453.48,Z 261.619,A -85,B 0,C 180,E1 -8224.988,E2 -8224.988} C_VEL
LIN {X 0,Y 453.462,Z 261.619,A -85,B 0,C 180,E1 -8228.311,E2 -8228.311} C_VEL
LIN {X 0,Y 453.491,Z 261.619,A -85,B 0,C 180,E1 -8230.608,E2 -8230.608} C_VEL
LIN {X 0,Y 453.459,Z 261.614,A -85,B 0,C 180,E1 -8233.244,E2 -8233.244} C_VEL
LIN {X 0,Y 453.462,Z 261.623,A -85,B 0,C 180,E1 -8235.778,E2 -8235.778} C_VEL
LIN {X 0,Y 453.511,Z 261.604,A -85,B 0,C 180,E1 -8239.405,E2 -8239.405} C_VEL
LIN {X 0,Y 453.471,Z 261.622,A -85,B 0,C 180,E1 -8242.222,E2 -8242.222} C_VEL
LIN {X 0,Y 453.483,Z 261.607,A -85,B 0,C 180,E1 -8245.222,E2 -8245.222} C_VEL
LIN {X 0,Y 453.462,Z 261.61,A -85,B 0,C 180,E1 -8248.474,E2 -8248.474} C_VEL
LIN {X 0,Y 453.509,Z 261.621,A -85,B 0,C 180,E1 -8251.288,E2 -8251.288} C_VEL
LIN {X 0,Y 453.517,Z 261.608,A -85,B 0,C 180,E1 -8254.284,E2 -8254.284} C_VEL
LIN {X 0,Y 453.471,Z 261.623,A -85,B 0,C 180,E1 -8257.204,E2 -8257.204} C_VEL
LIN {X 0,Y 453.496,Z 261.612,A -85,B 0,C 180,E1 -8260.066,E2 -8260.066} C_VEL
LIN {X 0,Y 453.499,Z 261.621,A -85,B 0,C 180,E1 -8262.875,E2 -8262.875} C_VEL
LIN {X 0,Y 453.505,Z 261.61,A -85,B 0,C 180,E1 -8265.643,E2 -8265.643} C_VEL
LIN {X 0,Y 453.553,Z 261.613,A -85,B 0,C 180,E1 -8268.379,E2 -8268.379} C_VEL
LIN {X 0,Y 453.643,Z 261.591,A -85,B 0,C 180,E1 -8271.985,E2 -8271.985} C_VEL
LIN {X 0,Y 453.666,Z 261.602,A -85,B 0,C 180,E1 -8274.667,E2 -8274.667} C_VEL
LIN {X 0,Y 453.757,Z 261.574,A -85,B 0,C 180,E1 -8277.337,E2 -8277.337} C_VEL
LIN {X 0,Y 453.815,Z 261.577,A -85,B 0,C 180,E1 -8280,E2 -8280} C_VEL
LIN {X 0,Y 453.757,Z 261.582,A -85,B 0,C 180,E1 -8282.663,E2 -8282.663} C_VEL
LIN {X 0,Y 453.669,Z 261.597,A -85,B 0,C 180,E1 -8286.225,E2 -8286.225} C_VEL
LIN {X 0,Y 453.584,Z 261.602,A -85,B 0,C 180,E1 -8288.913,E2 -8288.913} C_VEL
LIN {X 0,Y 453.554,Z 261.615,A -85,B 0,C 180,E1 -8292.529,E2 -8292.529} C_VEL
LIN {X 0,Y 453.536,Z 261.609,A -85,B 0,C 180,E1 -8296.196,E2 -8296.196} C_VEL
LIN {X 0,Y 453.511,Z 261.615,A -85,B 0,C 180,E1 -8299.041,E2 -8299.041} C_VEL
LIN {X 0,Y 453.469,Z 261.619,A -85,B 0,C 180,E1 -8301.836,E2 -8301.836} C_VEL
LIN {X 0,Y 453.506,Z 261.617,A -85,B 0,C 180,E1 -8304.735,E2 -8304.735} C_VEL
LIN {X 0,Y 453.531,Z 261.612,A -85,B 0,C 180,E1 -8307.962,E2 -8307.962} C_VEL
LIN {X 0,Y 453.476,Z 261.619,A -85,B 0,C 180,E1 -8310.76,E2 -8310.76} C_VEL
LIN {X 0,Y 453.471,Z 261.6,A -85,B 0,C 180,E1 -8313.913,E2 -8313.913} C_VEL
LIN {X 0,Y 453.464,Z 261.618,A -85,B 0,C 180,E1 -8317.189,E2 -8317.189} C_VEL
LIN {X 0,Y 453.511,Z 261.619,A -85,B 0,C 180,E1 -8319.448,E2 -8319.448} C_VEL
LIN {X 0,Y 453.458,Z 261.623,A -85,B 0,C 180,E1 -8322.996,E2 -8322.996} C_VEL
LIN {X 0,Y 453.472,Z 261.625,A -85,B 0,C 180,E1 -8325.781,E2 -8325.781} C_VEL
LIN {X 0,Y 453.492,Z 261.606,A -85,B 0,C 180,E1 -8328.212,E2 -8328.212} C_VEL
LIN {X 0,Y 453.527,Z 261.615,A -85,B 0,C 180,E1 -8330.788,E2 -8330.788} C_VEL
LIN {X 0,Y 453.451,Z 261.625,A -85,B 0,C 180,E1 -8333.918,E2 -8333.918} C_VEL
LIN {X 0,Y 453.48,Z 261.618,A -85,B 0,C 180,E1 -8337.152,E2 -8337.152} C_VEL
LIN {X 0,Y 453.472,Z 261.597,A -85,B 0,C 180,E1 -8340.269,E2 -8340.269} C_VEL
LIN {X 0,Y 453.6,Z 261.781,A -85,B 0,C 180,E1 -8342.553,E2 -8342.553} C_VEL
LIN {X 0,Y 456.129,Z 273.701,A -85,B 0,C 180,E1 -8344.926,E2 -8344.926} C_VEL
LIN {X 0,Y 456.853,Z 279.111,A -85,B 0,C 180,E1 -8345.943,E2 -8345.943} C_VEL
LIN {X 0,Y 455.873,Z 295.025,A -85,B 0,C 180,E1 -8348.696,E2 -8348.696} C_VEL
LIN {X 0,Y 457.979,Z 305.7,A -85,B 0,C 180,E1 -8349.006,E2 -8349.006} C_VEL
LIN {X 0,Y 460.153,Z 317.767,A -85,B 0,C 180,E1 -8349.306,E2 -8349.306} C_VEL
LIN {X 0,Y 458.885,Z 430.308,A -85,B 0,C 180,E1 -8351.095,E2 -8351.095} C_VEL
LIN {X 0,Y 458.49,Z 444.258,A -85,B 0,C 180,E1 -8351.454,E2 -8351.454} C_VEL
LIN {X 0,Y 457.976,Z 457.283,A -85,B 0,C 180,E1 -8351.954,E2 -8351.954} C_VEL
LIN {X 0,Y 457.329,Z 471.125,A -85,B 0,C 180,E1 -8352.672,E2 -8352.672} C_VEL
LIN {X 0,Y 456.564,Z 484.377,A -85,B 0,C 180,E1 -8353.57,E2 -8353.57} C_VEL
LIN {X 0,Y 455.717,Z 496.272,A -85,B 0,C 180,E1 -8354.572,E2 -8354.572} C_VEL
LIN {X 0,Y 454.992,Z 507.137,A -85,B 0,C 180,E1 -8355.692,E2 -8355.692} C_VEL
LIN {X 0,Y 454.279,Z 518.121,A -85,B 0,C 180,E1 -8357.072,E2 -8357.072} C_VEL
LIN {X 0,Y 453.789,Z 526.736,A -85,B 0,C 180,E1 -8358.385,E2 -8358.385} C_VEL
LIN {X 0,Y 453.222,Z 535.228,A -85,B 0,C 180,E1 -8359.954,E2 -8359.954} C_VEL
LIN {X 0,Y 452.889,Z 542.072,A -85,B 0,C 180,E1 -8361.523,E2 -8361.523} C_VEL
LIN {X 0,Y 452.664,Z 546.789,A -85,B 0,C 180,E1 -8362.865,E2 -8362.865} C_VEL
LIN {X 0,Y 452.579,Z 551.675,A -85,B 0,C 180,E1 -8364.654,E2 -8364.654} C_VEL
LIN {X 0,Y 452.446,Z 555.072,A -85,B 0,C 180,E1 -8366.438,E2 -8366.438} C_VEL
LIN {X 0,Y 452.43,Z 557.081,A -85,B 0,C 180,E1 -8368.22,E2 -8368.22} C_VEL
LIN {X 0,Y 452.405,Z 557.747,A -85,B 0,C 180,E1 -8370,E2 -8370} C_VEL
LIN {X 0,Y 452.43,Z 557.081,A -85,B 0,C 180,E1 -8371.78,E2 -8371.78} C_VEL
LIN {X 0,Y 452.446,Z 555.073,A -85,B 0,C 180,E1 -8373.562,E2 -8373.562} C_VEL
LIN {X 0,Y 452.585,Z 551.674,A -85,B 0,C 180,E1 -8375.346,E2 -8375.346} C_VEL
LIN {X 0,Y 452.662,Z 546.781,A -85,B 0,C 180,E1 -8377.135,E2 -8377.135} C_VEL
LIN {X 0,Y 452.968,Z 540.25,A -85,B 0,C 180,E1 -8378.926,E2 -8378.926} C_VEL
LIN {X 0,Y 453.332,Z 532.983,A -85,B 0,C 180,E1 -8380.495,E2 -8380.495} C_VEL
LIN {X 0,Y 453.962,Z 523.982,A -85,B 0,C 180,E1 -8382.064,E2 -8382.064} C_VEL
LIN {X 0,Y 454.533,Z 514.535,A -85,B 0,C 180,E1 -8383.411,E2 -8383.411} C_VEL
LIN {X 0,Y 455.212,Z 504.075,A -85,B 0,C 180,E1 -8384.644,E2 -8384.644} C_VEL
LIN {X 0,Y 455.978,Z 492.533,A -85,B 0,C 180,E1 -8385.762,E2 -8385.762} C_VEL
LIN {X 0,Y 456.82,Z 479.728,A -85,B 0,C 180,E1 -8386.766,E2 -8386.766} C_VEL
LIN {X 0,Y 457.604,Z 466.396,A -85,B 0,C 180,E1 -8387.589,E2 -8387.589} C_VEL
LIN {X 0,Y 458.128,Z 453.297,A -85,B 0,C 180,E1 -8388.214,E2 -8388.214} C_VEL
LIN {X 0,Y 458.654,Z 439.573,A -85,B 0,C 180,E1 -8388.684,E2 -8388.684} C_VEL
LIN {X 0,Y 458.957,Z 425.608,A -85,B 0,C 180,E1 -8388.989,E2 -8388.989} C_VEL
LIN {X 0,Y 460.082,Z 317.241,A -85,B 0,C 180,E1 -8390.702,E2 -8390.702} C_VEL
LIN {X 0,Y 455.878,Z 295.272,A -85,B 0,C 180,E1 -8391.282,E2 -8391.282} C_VEL
LIN {X 0,Y 456.142,Z 290.353,A -85,B 0,C 180,E1 -8392.082,E2 -8392.082} C_VEL
LIN {X 0,Y 456.844,Z 277.734,A -85,B 0,C 180,E1 -8394.3,E2 -8394.3} C_VEL
LIN {X 0,Y 454.454,Z 265.618,A -85,B 0,C 180,E1 -8396.645,E2 -8396.645} C_VEL
LIN {X 0,Y 453.588,Z 261.69,A -85,B 0,C 180,E1 -8397.479,E2 -8397.479} C_VEL
LIN {X 0,Y 453.475,Z 261.607,A -85,B 0,C 180,E1 -8400.759,E2 -8400.759} C_VEL
LIN {X 0,Y 453.474,Z 261.615,A -85,B 0,C 180,E1 -8403.912,E2 -8403.912} C_VEL
LIN {X 0,Y 453.449,Z 261.617,A -85,B 0,C 180,E1 -8407.189,E2 -8407.189} C_VEL
LIN {X 0,Y 453.486,Z 261.62,A -85,B 0,C 180,E1 -8409.449,E2 -8409.449} C_VEL
LIN {X 0,Y 453.476,Z 261.609,A -85,B 0,C 180,E1 -8411.935,E2 -8411.935} C_VEL
LIN {X 0,Y 453.483,Z 261.618,A -85,B 0,C 180,E1 -8415.47,E2 -8415.47} C_VEL
LIN {X 0,Y 453.475,Z 261.625,A -85,B 0,C 180,E1 -8418.209,E2 -8418.209} C_VEL
LIN {X 0,Y 453.51,Z 261.617,A -85,B 0,C 180,E1 -8420.789,E2 -8420.789} C_VEL
LIN {X 0,Y 453.451,Z 261.613,A -85,B 0,C 180,E1 -8423.917,E2 -8423.917} C_VEL
LIN {X 0,Y 453.477,Z 261.608,A -85,B 0,C 180,E1 -8427.151,E2 -8427.151} C_VEL
LIN {X 0,Y 453.508,Z 261.62,A -85,B 0,C 180,E1 -8430.271,E2 -8430.271} C_VEL
LIN {X 0,Y 453.507,Z 261.611,A -85,B 0,C 180,E1 -8433.294,E2 -8433.294} C_VEL
LIN {X 0,Y 453.497,Z 261.617,A -85,B 0,C 180,E1 -8436.238,E2 -8436.238} C_VEL
LIN {X 0,Y 453.475,Z 261.617,A -85,B 0,C 180,E1 -8439.117,E2 -8439.117} C_VEL
LIN {X 0,Y 453.504,Z 261.617,A -85,B 0,C 180,E1 -8441.944,E2 -8441.944} C_VEL
LIN {X 0,Y 453.532,Z 261.609,A -85,B 0,C 180,E1 -8444.726,E2 -8444.726} C_VEL
LIN {X 0,Y 453.551,Z 261.606,A -85,B 0,C 180,E1 -8448.379,E2 -8448.379} C_VEL
LIN {X 0,Y 453.644,Z 261.602,A -85,B 0,C 180,E1 -8451.985,E2 -8451.985} C_VEL
LIN {X 0,Y 453.663,Z 261.592,A -85,B 0,C 180,E1 -8454.667,E2 -8454.667} C_VEL
LIN {X 0,Y 453.757,Z 261.582,A -85,B 0,C 180,E1 -8457.337,E2 -8457.337} C_VEL
LIN {X 0,Y 453.815,Z 261.577,A -85,B 0,C 180,E1 -8460,E2 -8460} C_VEL
LIN {X 0,Y 453.758,Z 261.573,A -85,B 0,C 180,E1 -8462.663,E2 -8462.663} C_VEL
LIN {X 0,Y 453.672,Z 261.595,A -85,B 0,C 180,E1 -8466.225,E2 -8466.225} C_VEL
LIN {X 0,Y 453.584,Z 261.6,A -85,B 0,C 180,E1 -8468.914,E2 -8468.914} C_VEL
LIN {X 0,Y 453.556,Z 261.61,A -85,B 0,C 180,E1 -8472.529,E2 -8472.529} C_VEL
LIN {X 0,Y 453.537,Z 261.608,A -85,B 0,C 180,E1 -8476.196,E2 -8476.196} C_VEL
LIN {X 0,Y 453.513,Z 261.62,A -85,B 0,C 180,E1 -8479.041,E2 -8479.041} C_VEL
LIN {X 0,Y 453.469,Z 261.618,A -85,B 0,C 180,E1 -8481.837,E2 -8481.837} C_VEL
LIN {X 0,Y 453.507,Z 261.619,A -85,B 0,C 180,E1 -8484.735,E2 -8484.735} C_VEL
LIN {X 0,Y 453.533,Z 261.612,A -85,B 0,C 180,E1 -8487.962,E2 -8487.962} C_VEL
LIN {X 0,Y 453.478,Z 261.619,A -85,B 0,C 180,E1 -8490.76,E2 -8490.76} C_VEL
LIN {X 0,Y 453.472,Z 261.597,A -85,B 0,C 180,E1 -8493.913,E2 -8493.913} C_VEL
LIN {X 0,Y 453.466,Z 261.625,A -85,B 0,C 180,E1 -8497.189,E2 -8497.189} C_VEL
LIN {X 0,Y 453.523,Z 261.609,A -85,B 0,C 180,E1 -8499.447,E2 -8499.447} C_VEL
LIN {X 0,Y 453.474,Z 261.602,A -85,B 0,C 180,E1 -8501.936,E2 -8501.936} C_VEL
LIN {X 0,Y 453.488,Z 261.618,A -85,B 0,C 180,E1 -8505.471,E2 -8505.471} C_VEL
LIN {X 0,Y 453.479,Z 261.608,A -85,B 0,C 180,E1 -8508.21,E2 -8508.21} C_VEL
LIN {X 0,Y 453.513,Z 261.617,A -85,B 0,C 180,E1 -8510.791,E2 -8510.791} C_VEL
LIN {X 0,Y 453.455,Z 261.624,A -85,B 0,C 180,E1 -8513.918,E2 -8513.918} C_VEL
LIN {X 0,Y 453.482,Z 261.622,A -85,B 0,C 180,E1 -8517.152,E2 -8517.152} C_VEL
LIN {X 0,Y 453.475,Z 261.623,A -85,B 0,C 180,E1 -8520.269,E2 -8520.269} C_VEL
LIN {X 0,Y 453.504,Z 261.616,A -85,B 0,C 180,E1 -8523.294,E2 -8523.294} C_VEL
LIN {X 0,Y 453.559,Z 261.86,A -85,B 0,C 180,E1 -8523.792,E2 -8523.792} C_VEL
LIN {X 0,Y 456.437,Z 275.732,A -85,B 0,C 180,E1 -8526.642,E2 -8526.642} C_VEL
LIN {X 0,Y 456.384,Z 280.375,A -85,B 0,C 180,E1 -8527.512,E2 -8527.512} C_VEL
LIN {X 0,Y 456.011,Z 287.473,A -85,B 0,C 180,E1 -8528.767,E2 -8528.767} C_VEL
LIN {X 0,Y 460.224,Z 308.886,A -85,B 0,C 180,E1 -8529.345,E2 -8529.345} C_VEL
LIN {X 0,Y 459.538,Z 377.877,A -85,B 0,C 180,E1 -8530.438,E2 -8530.438} C_VEL
LIN {X 0,Y 458.855,Z 383.724,A -85,B 0,C 180,E1 -8530.503,E2 -8530.503} C_VEL
LIN {X 0,Y 453.151,Z 402.736,A -85,B 0,C 180,E1 -8530.559,E2 -8530.559} C_VEL
LIN {X 0,Y 452.399,Z 408.586,A -85,B 0,C 180,E1 -8530.622,E2 -8530.622} C_VEL
LIN {X 0,Y 452.073,Z 427.75,A -85,B 0,C 180,E1 -8530.978,E2 -8530.978} C_VEL
LIN {X 0,Y 451.55,Z 442.419,A -85,B 0,C 180,E1 -8531.441,E2 -8531.441} C_VEL
LIN {X 0,Y 451.063,Z 455.463,A -85,B 0,C 180,E1 -8532.035,E2 -8532.035} C_VEL
LIN {X 0,Y 450.384,Z 467.674,A -85,B 0,C 180,E1 -8532.754,E2 -8532.754} C_VEL
LIN {X 0,Y 449.637,Z 479.917,A -85,B 0,C 180,E1 -8533.66,E2 -8533.66} C_VEL
LIN {X 0,Y 448.844,Z 491.129,A -85,B 0,C 180,E1 -8534.679,E2 -8534.679} C_VEL
LIN {X 0,Y 447.984,Z 502.402,A -85,B 0,C 180,E1 -8535.927,E2 -8535.927} C_VEL
LIN {X 0,Y 447.294,Z 512.467,A -85,B 0,C 180,E1 -8537.293,E2 -8537.293} C_VEL
LIN {X 0,Y 446.743,Z 520.823,A -85,B 0,C 180,E1 -8538.659,E2 -8538.659} C_VEL
LIN {X 0,Y 446.202,Z 528.805,A -85,B 0,C 180,E1 -8540.252,E2 -8540.252} C_VEL
LIN {X 0,Y 445.833,Z 535.229,A -85,B 0,C 180,E1 -8541.844,E2 -8541.844} C_VEL
LIN {X 0,Y 445.598,Z 540.927,A -85,B 0,C 180,E1 -8543.661,E2 -8543.661} C_VEL
LIN {X 0,Y 445.426,Z 545.07,A -85,B 0,C 180,E1 -8545.475,E2 -8545.475} C_VEL
LIN {X 0,Y 445.433,Z 547.78,A -85,B 0,C 180,E1 -8547.287,E2 -8547.287} C_VEL
LIN {X 0,Y 445.313,Z 549.142,A -85,B 0,C 180,E1 -8549.096,E2 -8549.096} C_VEL
LIN {X 0,Y 445.313,Z 549.18,A -85,B 0,C 180,E1 -8550.904,E2 -8550.904} C_VEL
LIN {X 0,Y 445.432,Z 547.891,A -85,B 0,C 180,E1 -8552.713,E2 -8552.713} C_VEL
LIN {X 0,Y 445.425,Z 545.247,A -85,B 0,C 180,E1 -8554.525,E2 -8554.525} C_VEL
LIN {X 0,Y 445.618,Z 541.178,A -85,B 0,C 180,E1 -8556.338,E2 -8556.338} C_VEL
LIN {X 0,Y 445.827,Z 535.558,A -85,B 0,C 180,E1 -8558.156,E2 -8558.156} C_VEL
LIN {X 0,Y 446.194,Z 529.211,A -85,B 0,C 180,E1 -8559.748,E2 -8559.748} C_VEL
LIN {X 0,Y 446.708,Z 521.32,A -85,B 0,C 180,E1 -8561.341,E2 -8561.341} C_VEL
LIN {X 0,Y 447.234,Z 513.066,A -85,B 0,C 180,E1 -8562.709,E2 -8562.709} C_VEL
LIN {X 0,Y 447.951,Z 503.119,A -85,B 0,C 180,E1 -8564.074,E2 -8564.074} C_VEL
LIN {X 0,Y 448.757,Z 492.049,A -85,B 0,C 180,E1 -8565.324,E2 -8565.324} C_VEL
LIN {X 0,Y 449.541,Z 481.028,A -85,B 0,C 180,E1 -8566.344,E2 -8566.344} C_VEL
LIN {X 0,Y 450.325,Z 469.067,A -85,B 0,C 180,E1 -8567.248,E2 -8567.248} C_VEL
LIN {X 0,Y 451.028,Z 455.832,A -85,B 0,C 180,E1 -8568.042,E2 -8568.042} C_VEL
LIN {X 0,Y 451.609,Z 442.12,A -85,B 0,C 180,E1 -8568.662,E2 -8568.662} C_VEL
LIN {X 0,Y 452.122,Z 427.854,A -85,B 0,C 180,E1 -8569.111,E2 -8569.111} C_VEL
LIN {X 0,Y 452.421,Z 407.969,A -85,B 0,C 180,E1 -8569.481,E2 -8569.481} C_VEL
LIN {X 0,Y 453.563,Z 309.589,A -85,B 0,C 180,E1 -8571.057,E2 -8571.057} C_VEL
LIN {X 0,Y 449.168,Z 287.524,A -85,B 0,C 180,E1 -8571.669,E2 -8571.669} C_VEL
LIN {X 0,Y 449.688,Z 278.835,A -85,B 0,C 180,E1 -8573.242,E2 -8573.242} C_VEL
LIN {X 0,Y 448.05,Z 269.933,A -85,B 0,C 180,E1 -8575.056,E2 -8575.056} C_VEL
LIN {X 0,Y 446.502,Z 262.586,A -85,B 0,C 180,E1 -8576.653,E2 -8576.653} C_VEL
LIN {X 0,Y 446.448,Z 262.49,A -85,B 0,C 180,E1 -8579.209,E2 -8579.209} C_VEL
LIN {X 0,Y 446.421,Z 262.502,A -85,B 0,C 180,E1 -8582.361,E2 -8582.361} C_VEL
LIN {X 0,Y 446.419,Z 262.506,A -85,B 0,C 180,E1 -8585.625,E2 -8585.625} C_VEL
LIN {X 0,Y 446.457,Z 262.493,A -85,B 0,C 180,E1 -8589.025,E2 -8589.025} C_VEL
LIN {X 0,Y 446.433,Z 262.484,A -85,B 0,C 180,E1 -8592.277,E2 -8592.277} C_VEL
LIN {X 0,Y 446.45,Z 262.498,A -85,B 0,C 180,E1 -8595.103,E2 -8595.103} C_VEL
LIN {X 0,Y 446.431,Z 262.479,A -85,B 0,C 180,E1 -8598.609,E2 -8598.609} C_VEL
LIN {X 0,Y 446.468,Z 262.492,A -85,B 0,C 180,E1 -8600.975,E2 -8600.975} C_VEL
LIN {X 0,Y 446.416,Z 262.496,A -85,B 0,C 180,E1 -8604.373,E2 -8604.373} C_VEL
LIN {X 0,Y 446.417,Z 262.484,A -85,B 0,C 180,E1 -8607.638,E2 -8607.638} C_VEL
LIN {X 0,Y 446.463,Z 262.497,A -85,B 0,C 180,E1 -8610.792,E2 -8610.792} C_VEL
LIN {X 0,Y 446.471,Z 262.485,A -85,B 0,C 180,E1 -8613.848,E2 -8613.848} C_VEL
LIN {X 0,Y 446.422,Z 262.504,A -85,B 0,C 180,E1 -8616.823,E2 -8616.823} C_VEL
LIN {X 0,Y 446.436,Z 262.491,A -85,B 0,C 180,E1 -8619.737,E2 -8619.737} C_VEL
LIN {X 0,Y 446.456,Z 262.499,A -85,B 0,C 180,E1 -8622.597,E2 -8622.597} C_VEL
LIN {X 0,Y 446.462,Z 262.488,A -85,B 0,C 180,E1 -8625.412,E2 -8625.412} C_VEL
LIN {X 0,Y 446.51,Z 262.488,A -85,B 0,C 180,E1 -8628.193,E2 -8628.193} C_VEL
LIN {X 0,Y 446.591,Z 262.469,A -85,B 0,C 180,E1 -8631.858,E2 -8631.858} C_VEL
LIN {X 0,Y 446.64,Z 262.478,A -85,B 0,C 180,E1 -8634.582,E2 -8634.582} C_VEL
LIN {X 0,Y 446.701,Z 262.452,A -85,B 0,C 180,E1 -8637.295,E2 -8637.295} C_VEL
LIN {X 0,Y 446.785,Z 262.453,A -85,B 0,C 180,E1 -8640,E2 -8640} C_VEL
LIN {X 0,Y 446.701,Z 262.46,A -85,B 0,C 180,E1 -8642.705,E2 -8642.705} C_VEL
LIN {X 0,Y 446.638,Z 262.474,A -85,B 0,C 180,E1 -8646.324,E2 -8646.324} C_VEL
LIN {X 0,Y 446.53,Z 262.48,A -85,B 0,C 180,E1 -8649.055,E2 -8649.055} C_VEL
LIN {X 0,Y 446.513,Z 262.49,A -85,B 0,C 180,E1 -8652.73,E2 -8652.73} C_VEL
LIN {X 0,Y 446.487,Z 262.487,A -85,B 0,C 180,E1 -8656.228,E2 -8656.228} C_VEL
LIN {X 0,Y 446.461,Z 262.494,A -85,B 0,C 180,E1 -8659.304,E2 -8659.304} C_VEL
LIN {X 0,Y 446.41,Z 262.497,A -85,B 0,C 180,E1 -8662.2,E2 -8662.2} C_VEL
LIN {X 0,Y 446.45,Z 262.495,A -85,B 0,C 180,E1 -8665.153,E2 -8665.153} C_VEL
LIN {X 0,Y 446.477,Z 262.492,A -85,B 0,C 180,E1 -8668.179,E2 -8668.179} C_VEL
LIN {X 0,Y 446.424,Z 262.498,A -85,B 0,C 180,E1 -8671.3,E2 -8671.3} C_VEL
LIN {X 0,Y 446.423,Z 262.475,A -85,B 0,C 180,E1 -8674.524,E2 -8674.524} C_VEL
LIN {X 0,Y 446.425,Z 262.503,A -85,B 0,C 180,E1 -8678.082,E2 -8678.082} C_VEL
LIN {X 0,Y 446.421,Z 262.495,A -85,B 0,C 180,E1 -8680.918,E2 -8680.918} C_VEL
LIN {X 0,Y 446.397,Z 262.503,A -85,B 0,C 180,E1 -8683.847,E2 -8683.847} C_VEL
LIN {X 0,Y 446.443,Z 262.495,A -85,B 0,C 180,E1 -8686.398,E2 -8686.398} C_VEL
LIN {X 0,Y 446.465,Z 262.493,A -85,B 0,C 180,E1 -8689.806,E2 -8689.806} C_VEL
LIN {X 0,Y 446.429,Z 262.493,A -85,B 0,C 180,E1 -8692.124,E2 -8692.124} C_VEL
LIN {X 0,Y 446.426,Z 262.499,A -85,B 0,C 180,E1 -8695.478,E2 -8695.478} C_VEL
LIN {X 0,Y 446.414,Z 262.497,A -85,B 0,C 180,E1 -8698.7,E2 -8698.7} C_VEL
LIN {X 0,Y 446.503,Z 262.551,A -85,B 0,C 180,E1 -8702.206,E2 -8702.206} C_VEL
LIN {X 0,Y 447.218,Z 265.586,A -85,B 0,C 180,E1 -8702.889,E2 -8702.889} C_VEL
LIN {X 0,Y 449.691,Z 277.435,A -85,B 0,C 180,E1 -8705.239,E2 -8705.239} C_VEL
LIN {X 0,Y 449.842,Z 281.733,A -85,B 0,C 180,E1 -8706.034,E2 -8706.034} C_VEL
LIN {X 0,Y 449.064,Z 295.023,A -85,B 0,C 180,E1 -8708.361,E2 -8708.361} C_VEL
LIN {X 0,Y 453.408,Z 318.142,A -85,B 0,C 180,E1 -8708.991,E2 -8708.991} C_VEL
LIN {X 0,Y 452.489,Z 409.66,A -85,B 0,C 180,E1 -8710.463,E2 -8710.463} C_VEL
LIN {X 0,Y 452.09,Z 434.123,A -85,B 0,C 180,E1 -8710.888,E2 -8710.888} C_VEL
LIN {X 0,Y 451.589,Z 448.215,A -85,B 0,C 180,E1 -8711.308,E2 -8711.308} C_VEL
LIN {X 0,Y 450.985,Z 462.233,A -85,B 0,C 180,E1 -8711.916,E2 -8711.916} C_VEL
LIN {X 0,Y 450.258,Z 475.222,A -85,B 0,C 180,E1 -8712.666,E2 -8712.666} C_VEL
LIN {X 0,Y 449.521,Z 487.168,A -85,B 0,C 180,E1 -8713.539,E2 -8713.539} C_VEL
LIN {X 0,Y 448.7,Z 498.558,A -85,B 0,C 180,E1 -8714.558,E2 -8714.558} C_VEL
LIN {X 0,Y 447.943,Z 509.025,A -85,B 0,C 180,E1 -8715.694,E2 -8715.694} C_VEL
LIN {X 0,Y 447.294,Z 518.622,A -85,B 0,C 180,E1 -8716.947,E2 -8716.947} C_VEL
LIN {X 0,Y 446.692,Z 528.027,A -85,B 0,C 180,E1 -8718.428,E2 -8718.428} C_VEL
LIN {X 0,Y 446.126,Z 536.25,A -85,B 0,C 180,E1 -8720.021,E2 -8720.021} C_VEL
LIN {X 0,Y 445.825,Z 542.006,A -85,B 0,C 180,E1 -8721.387,E2 -8721.387} C_VEL
LIN {X 0,Y 445.59,Z 546.722,A -85,B 0,C 180,E1 -8722.751,E2 -8722.751} C_VEL
LIN {X 0,Y 445.491,Z 551.609,A -85,B 0,C 180,E1 -8724.569,E2 -8724.569} C_VEL
LIN {X 0,Y 445.345,Z 555.005,A -85,B 0,C 180,E1 -8726.381,E2 -8726.381} C_VEL
LIN {X 0,Y 445.349,Z 557.015,A -85,B 0,C 180,E1 -8728.191,E2 -8728.191} C_VEL
LIN {X 0,Y 445.314,Z 557.68,A -85,B 0,C 180,E1 -8730,E2 -8730} C_VEL
LIN {X 0,Y 445.349,Z 557.015,A -85,B 0,C 180,E1 -8731.809,E2 -8731.809} C_VEL
LIN {X 0,Y 445.346,Z 555.006,A -85,B 0,C 180,E1 -8733.619,E2 -8733.619} C_VEL
LIN {X 0,Y 445.498,Z 551.607,A -85,B 0,C 180,E1 -8735.431,E2 -8735.431} C_VEL
LIN {X 0,Y 445.589,Z 546.713,A -85,B 0,C 180,E1 -8737.249,E2 -8737.249} C_VEL
LIN {X 0,Y 445.924,Z 540.183,A -85,B 0,C 180,E1 -8739.068,E2 -8739.068} C_VEL
LIN {X 0,Y 446.324,Z 532.915,A -85,B 0,C 180,E1 -8740.662,E2 -8740.662} C_VEL
LIN {X 0,Y 446.97,Z 523.914,A -85,B 0,C 180,E1 -8742.255,E2 -8742.255} C_VEL
LIN {X 0,Y 447.589,Z 514.466,A -85,B 0,C 180,E1 -8743.623,E2 -8743.623} C_VEL
LIN {X 0,Y 448.312,Z 504.006,A -85,B 0,C 180,E1 -8744.874,E2 -8744.874} C_VEL
LIN {X 0,Y 449.098,Z 492.463,A -85,B 0,C 180,E1 -8746.01,E2 -8746.01} C_VEL
LIN {X 0,Y 449.927,Z 481.241,A -85,B 0,C 180,E1 -8746.913,E2 -8746.913} C_VEL
LIN {X 0,Y 450.705,Z 468.134,A -85,B 0,C 180,E1 -8747.761,E2 -8747.761} C_VEL
LIN {X 0,Y 451.344,Z 454.526,A -85,B 0,C 180,E1 -8748.438,E2 -8748.438} C_VEL
LIN {X 0,Y 451.916,Z 440.413,A -85,B 0,C 180,E1 -8748.943,E2 -8748.943} C_VEL
LIN {X 0,Y 452.229,Z 427.05,A -85,B 0,C 180,E1 -8749.254,E2 -8749.254} C_VEL
LIN {X 0,Y 453.492,Z 319.365,A -85,B 0,C 180,E1 -8750.98,E2 -8750.98} C_VEL
LIN {X 0,Y 450.648,Z 303.34,A -85,B 0,C 180,E1 -8751.387,E2 -8751.387} C_VEL
LIN {X 0,Y 449.023,Z 294.971,A -85,B 0,C 180,E1 -8751.641,E2 -8751.641} C_VEL
LIN {X 0,Y 449.96,Z 280.355,A -85,B 0,C 180,E1 -8754.204,E2 -8754.204} C_VEL
LIN {X 0,Y 449.188,Z 274.977,A -85,B 0,C 180,E1 -8755.236,E2 -8755.236} C_VEL
LIN {X 0,Y 446.532,Z 262.667,A -85,B 0,C 180,E1 -8757.728,E2 -8757.728} C_VEL
LIN {X 0,Y 446.426,Z 262.477,A -85,B 0,C 180,E1 -8760.249,E2 -8760.249} C_VEL
LIN {X 0,Y 446.443,Z 262.49,A -85,B 0,C 180,E1 -8763.453,E2 -8763.453} C_VEL
LIN {X 0,Y 446.399,Z 262.496,A -85,B 0,C 180,E1 -8766.745,E2 -8766.745} C_VEL
LIN {X 0,Y 446.44,Z 262.496,A -85,B 0,C 180,E1 -8770.197,E2 -8770.197} C_VEL
LIN {X 0,Y 446.419,Z 262.498,A -85,B 0,C 180,E1 -8773.599,E2 -8773.599} C_VEL
LIN {X 0,Y 446.395,Z 262.505,A -85,B 0,C 180,E1 -8776.403,E2 -8776.403} C_VEL
LIN {X 0,Y 446.422,Z 262.494,A -85,B 0,C 180,E1 -8779.082,E2 -8779.082} C_VEL
LIN {X 0,Y 446.425,Z 262.503,A -85,B 0,C 180,E1 -8781.918,E2 -8781.918} C_VEL
LIN {X 0,Y 446.424,Z 262.474,A -85,B 0,C 180,E1 -8785.477,E2 -8785.477} C_VEL
LIN {X 0,Y 446.424,Z 262.498,A -85,B 0,C 180,E1 -8788.7,E2 -8788.7} C_VEL
LIN {X 0,Y 446.478,Z 262.492,A -85,B 0,C 180,E1 -8791.821,E2 -8791.821} C_VEL
LIN {X 0,Y 446.451,Z 262.495,A -85,B 0,C 180,E1 -8794.847,E2 -8794.847} C_VEL
LIN {X 0,Y 446.441,Z 262.495,A -85,B 0,C 180,E1 -8798.245,E2 -8798.245} C_VEL
LIN {X 0,Y 446.45,Z 262.5,A -85,B 0,C 180,E1 -8801.649,E2 -8801.649} C_VEL
LIN {X 0,Y 446.5,Z 262.486,A -85,B 0,C 180,E1 -8804.48,E2 -8804.48} C_VEL
LIN {X 0,Y 446.509,Z 262.484,A -85,B 0,C 180,E1 -8808.193,E2 -8808.193} C_VEL
LIN {X 0,Y 446.592,Z 262.482,A -85,B 0,C 180,E1 -8811.858,E2 -8811.858} C_VEL
LIN {X 0,Y 446.638,Z 262.467,A -85,B 0,C 180,E1 -8814.583,E2 -8814.583} C_VEL
LIN {X 0,Y 446.701,Z 262.46,A -85,B 0,C 180,E1 -8817.295,E2 -8817.295} C_VEL
LIN {X 0,Y 446.785,Z 262.453,A -85,B 0,C 180,E1 -8820,E2 -8820} C_VEL
LIN {X 0,Y 446.702,Z 262.452,A -85,B 0,C 180,E1 -8822.705,E2 -8822.705} C_VEL
LIN {X 0,Y 446.64,Z 262.471,A -85,B 0,C 180,E1 -8826.324,E2 -8826.324} C_VEL
LIN {X 0,Y 446.53,Z 262.479,A -85,B 0,C 180,E1 -8829.056,E2 -8829.056} C_VEL
LIN {X 0,Y 446.516,Z 262.488,A -85,B 0,C 180,E1 -8832.73,E2 -8832.73} C_VEL
LIN {X 0,Y 446.489,Z 262.486,A -85,B 0,C 180,E1 -8836.228,E2 -8836.228} C_VEL
LIN {X 0,Y 446.462,Z 262.494,A -85,B 0,C 180,E1 -8839.304,E2 -8839.304} C_VEL
LIN {X 0,Y 446.411,Z 262.497,A -85,B 0,C 180,E1 -8842.2,E2 -8842.2} C_VEL
LIN {X 0,Y 446.451,Z 262.494,A -85,B 0,C 180,E1 -8845.153,E2 -8845.153} C_VEL
LIN {X 0,Y 446.478,Z 262.491,A -85,B 0,C 180,E1 -8848.179,E2 -8848.179} C_VEL
LIN {X 0,Y 446.414,Z 262.49,A -85,B 0,C 180,E1 -8851.301,E2 -8851.301} C_VEL
LIN {X 0,Y 446.425,Z 262.478,A -85,B 0,C 180,E1 -8854.524,E2 -8854.524} C_VEL
LIN {X 0,Y 446.43,Z 262.499,A -85,B 0,C 180,E1 -8858.083,E2 -8858.083} C_VEL
LIN {X 0,Y 446.439,Z 262.48,A -85,B 0,C 180,E1 -8860.921,E2 -8860.921} C_VEL
LIN {X 0,Y 446.398,Z 262.499,A -85,B 0,C 180,E1 -8863.847,E2 -8863.847} C_VEL
LIN {X 0,Y 446.418,Z 262.498,A -85,B 0,C 180,E1 -8866.401,E2 -8866.401} C_VEL
LIN {X 0,Y 446.449,Z 262.496,A -85,B 0,C 180,E1 -8869.804,E2 -8869.804} C_VEL
LIN {X 0,Y 446.408,Z 262.496,A -85,B 0,C 180,E1 -8872.122,E2 -8872.122} C_VEL
LIN {X 0,Y 446.429,Z 262.495,A -85,B 0,C 180,E1 -8875.478,E2 -8875.478} C_VEL
LIN {X 0,Y 446.415,Z 262.499,A -85,B 0,C 180,E1 -8878.7,E2 -8878.7} C_VEL
LIN {X 0,Y 446.485,Z 262.475,A -85,B 0,C 180,E1 -8881.822,E2 -8881.822} C_VEL
LIN {X 0,Y 446.501,Z 262.669,A -85,B 0,C 180,E1 -8883.486,E2 -8883.486} C_VEL
LIN {X 0,Y 449.235,Z 275.798,A -85,B 0,C 180,E1 -8886.245,E2 -8886.245} C_VEL
LIN {X 0,Y 449.661,Z 279.616,A -85,B 0,C 180,E1 -8887,E2 -8887} C_VEL
LIN {X 0,Y 449.145,Z 287.546,A -85,B 0,C 180,E1 -8888.426,E2 -8888.426} C_VEL
LIN {X 0,Y 453.509,Z 308.919,A -85,B 0,C 180,E1 -8889.024,E2 -8889.024} C_VEL
LIN {X 0,Y 452.399,Z 408.586,A -85,B 0,C 180,E1 -8890.622,E2 -8890.622} C_VEL
LIN {X 0,Y 451.668,Z 414.431,A -85,B 0,C 180,E1 -8890.685,E2 -8890.685} C_VEL
LIN {X 0,Y 448.846,Z 423.929,A -85,B 0,C 180,E1 -8890.737,E2 -8890.737} C_VEL
LIN {X 0,Y 445.929,Z 433.331,A -85,B 0,C 180,E1 -8890.86,E2 -8890.86} C_VEL
LIN {X 0,Y 445.009,Z 439.021,A -85,B 0,C 180,E1 -8891.021,E2 -8891.021} C_VEL
LIN {X 0,Y 444.49,Z 451.858,A -85,B 0,C 180,E1 -8891.565,E2 -8891.565} C_VEL
LIN {X 0,Y 443.807,Z 464.936,A -85,B 0,C 180,E1 -8892.3,E2 -8892.3} C_VEL
LIN {X 0,Y 442.997,Z 477.142,A -85,B 0,C 180,E1 -8893.171,E2 -8893.171} C_VEL
LIN {X 0,Y 442.134,Z 488.857,A -85,B 0,C 180,E1 -8894.204,E2 -8894.204} C_VEL
LIN {X 0,Y 441.225,Z 500.549,A -85,B 0,C 180,E1 -8895.471,E2 -8895.471} C_VEL
LIN {X 0,Y 440.478,Z 510.078,A -85,B 0,C 180,E1 -8896.726,E2 -8896.726} C_VEL
LIN {X 0,Y 439.974,Z 518.255,A -85,B 0,C 180,E1 -8898.015,E2 -8898.015} C_VEL
LIN {X 0,Y 439.322,Z 526.764,A -85,B 0,C 180,E1 -8899.632,E2 -8899.632} C_VEL
LIN {X 0,Y 438.877,Z 533.618,A -85,B 0,C 180,E1 -8901.25,E2 -8901.25} C_VEL
LIN {X 0,Y 438.614,Z 538.35,A -85,B 0,C 180,E1 -8902.635,E2 -8902.635} C_VEL
LIN {X 0,Y 438.467,Z 543.251,A -85,B 0,C 180,E1 -8904.481,E2 -8904.481} C_VEL
LIN {X 0,Y 438.291,Z 546.666,A -85,B 0,C 180,E1 -8906.323,E2 -8906.323} C_VEL
LIN {X 0,Y 438.341,Z 547.848,A -85,B 0,C 180,E1 -8907.243,E2 -8907.243} C_VEL
LIN {X 0,Y 438.229,Z 549.208,A -85,B 0,C 180,E1 -8909.081,E2 -8909.081} C_VEL
LIN {X 0,Y 438.229,Z 549.246,A -85,B 0,C 180,E1 -8910.919,E2 -8910.919} C_VEL
LIN {X 0,Y 438.341,Z 547.957,A -85,B 0,C 180,E1 -8912.757,E2 -8912.757} C_VEL
LIN {X 0,Y 438.352,Z 545.313,A -85,B 0,C 180,E1 -8914.598,E2 -8914.598} C_VEL
LIN {X 0,Y 438.545,Z 541.244,A -85,B 0,C 180,E1 -8916.441,E2 -8916.441} C_VEL
LIN {X 0,Y 438.771,Z 535.623,A -85,B 0,C 180,E1 -8918.288,E2 -8918.288} C_VEL
LIN {X 0,Y 439.175,Z 529.276,A -85,B 0,C 180,E1 -8919.906,E2 -8919.906} C_VEL
LIN {X 0,Y 439.73,Z 521.384,A -85,B 0,C 180,E1 -8921.524,E2 -8921.524} C_VEL
LIN {X 0,Y 440.326,Z 512.401,A -85,B 0,C 180,E1 -8923.027,E2 -8923.027} C_VEL
LIN {X 0,Y 441.031,Z 503.183,A -85,B 0,C 180,E1 -8924.3,E2 -8924.3} C_VEL
LIN {X 0,Y 441.875,Z 492.112,A -85,B 0,C 180,E1 -8925.568,E2 -8925.568} C_VEL
LIN {X 0,Y 442.716,Z 481.089,A -85,B 0,C 180,E1 -8926.603,E2 -8926.603} C_VEL
LIN {X 0,Y 443.627,Z 467.864,A -85,B 0,C 180,E1 -8927.603,E2 -8927.603} C_VEL
LIN {X 0,Y 444.295,Z 455.24,A -85,B 0,C 180,E1 -8928.359,E2 -8928.359} C_VEL
LIN {X 0,Y 444.914,Z 441.414,A -85,B 0,C 180,E1 -8928.984,E2 -8928.984} C_VEL
LIN {X 0,Y 445.458,Z 426.764,A -85,B 0,C 180,E1 -8929.438,E2 -8929.438} C_VEL
LIN {X 0,Y 445.818,Z 402.643,A -85,B 0,C 180,E1 -8929.871,E2 -8929.871} C_VEL
LIN {X 0,Y 446.893,Z 309.742,A -85,B 0,C 180,E1 -8931.384,E2 -8931.384} C_VEL
LIN {X 0,Y 442.334,Z 287.557,A -85,B 0,C 180,E1 -8932.024,E2 -8932.024} C_VEL
LIN {X 0,Y 442.781,Z 280.172,A -85,B 0,C 180,E1 -8933.378,E2 -8933.378} C_VEL
LIN {X 0,Y 440.866,Z 269.996,A -85,B 0,C 180,E1 -8935.493,E2 -8935.493} C_VEL
LIN {X 0,Y 439.445,Z 263.454,A -85,B 0,C 180,E1 -8936.955,E2 -8936.955} C_VEL
LIN {X 0,Y 439.381,Z 263.376,A -85,B 0,C 180,E1 -8939.725,E2 -8939.725} C_VEL
LIN {X 0,Y 439.371,Z 263.38,A -85,B 0,C 180,E1 -8942.945,E2 -8942.945} C_VEL
LIN {X 0,Y 439.372,Z 263.38,A -85,B 0,C 180,E1 -8946.286,E2 -8946.286} C_VEL
LIN {X 0,Y 439.41,Z 263.377,A -85,B 0,C 180,E1 -8949.85,E2 -8949.85} C_VEL
LIN {X 0,Y 439.382,Z 263.362,A -85,B 0,C 180,E1 -8952.627,E2 -8952.627} C_VEL
LIN {X 0,Y 439.398,Z 263.379,A -85,B 0,C 180,E1 -8955.27,E2 -8955.27} C_VEL
LIN {X 0,Y 439.393,Z 263.355,A -85,B 0,C 180,E1 -8958.741,E2 -8958.741} C_VEL
LIN {X 0,Y 439.387,Z 263.381,A -85,B 0,C 180,E1 -8961.604,E2 -8961.604} C_VEL
LIN {X 0,Y 439.395,Z 263.367,A -85,B 0,C 180,E1 -8964.843,E2 -8964.843} C_VEL
LIN {X 0,Y 439.368,Z 263.364,A -85,B 0,C 180,E1 -8968.139,E2 -8968.139} C_VEL
LIN {X 0,Y 439.419,Z 263.376,A -85,B 0,C 180,E1 -8971.326,E2 -8971.326} C_VEL
LIN {X 0,Y 439.398,Z 263.367,A -85,B 0,C 180,E1 -8974.415,E2 -8974.415} C_VEL
LIN {X 0,Y 439.357,Z 263.378,A -85,B 0,C 180,E1 -8977.424,E2 -8977.424} C_VEL
LIN {X 0,Y 439.433,Z 263.368,A -85,B 0,C 180,E1 -8980.662,E2 -8980.662} C_VEL
LIN {X 0,Y 439.454,Z 263.364,A -85,B 0,C 180,E1 -8984.224,E2 -8984.224} C_VEL
LIN {X 0,Y 439.476,Z 263.364,A -85,B 0,C 180,E1 -8988.001,E2 -8988.001} C_VEL
LIN {X 0,Y 439.539,Z 263.347,A -85,B 0,C 180,E1 -8991.726,E2 -8991.726} C_VEL
LIN {X 0,Y 439.615,Z 263.352,A -85,B 0,C 180,E1 -8994.496,E2 -8994.496} C_VEL
LIN {X 0,Y 439.627,Z 263.335,A -85,B 0,C 180,E1 -8998.168,E2 -8998.168} C_VEL
LIN {X 0,Y 439.756,Z 263.328,A -85,B 0,C 180,E1 -9000,E2 -9000} C_VEL
LIN {X 0,Y 439.648,Z 263.338,A -85,B 0,C 180,E1 -9002.749,E2 -9002.749} C_VEL
LIN {X 0,Y 439.609,Z 263.351,A -85,B 0,C 180,E1 -9006.425,E2 -9006.425} C_VEL
LIN {X 0,Y 439.491,Z 263.356,A -85,B 0,C 180,E1 -9009.202,E2 -9009.202} C_VEL
LIN {X 0,Y 439.457,Z 263.367,A -85,B 0,C 180,E1 -9012.938,E2 -9012.938} C_VEL
LIN {X 0,Y 439.439,Z 263.364,A -85,B 0,C 180,E1 -9016.349,E2 -9016.349} C_VEL
LIN {X 0,Y 439.394,Z 263.376,A -85,B 0,C 180,E1 -9019.627,E2 -9019.627} C_VEL
LIN {X 0,Y 439.357,Z 263.377,A -85,B 0,C 180,E1 -9022.576,E2 -9022.576} C_VEL
LIN {X 0,Y 439.398,Z 263.376,A -85,B 0,C 180,E1 -9025.585,E2 -9025.585} C_VEL
LIN {X 0,Y 439.418,Z 263.371,A -85,B 0,C 180,E1 -9028.673,E2 -9028.673} C_VEL
LIN {X 0,Y 439.376,Z 263.37,A -85,B 0,C 180,E1 -9032.034,E2 -9032.034} C_VEL
LIN {X 0,Y 439.39,Z 263.353,A -85,B 0,C 180,E1 -9035.341,E2 -9035.341} C_VEL
LIN {X 0,Y 439.384,Z 263.376,A -85,B 0,C 180,E1 -9038.595,E2 -9038.595} C_VEL
LIN {X 0,Y 439.383,Z 263.373,A -85,B 0,C 180,E1 -9041.257,E2 -9041.257} C_VEL
LIN {X 0,Y 439.398,Z 263.373,A -85,B 0,C 180,E1 -9044.73,E2 -9044.73} C_VEL
LIN {X 0,Y 439.408,Z 263.362,A -85,B 0,C 180,E1 -9047.798,E2 -9047.798} C_VEL
LIN {X 0,Y 439.447,Z 263.37,A -85,B 0,C 180,E1 -9050.231,E2 -9050.231} C_VEL
LIN {X 0,Y 439.373,Z 263.375,A -85,B 0,C 180,E1 -9053.714,E2 -9053.714} C_VEL
LIN {X 0,Y 439.37,Z 263.375,A -85,B 0,C 180,E1 -9057.055,E2 -9057.055} C_VEL
LIN {X 0,Y 439.38,Z 263.351,A -85,B 0,C 180,E1 -9060.275,E2 -9060.275} C_VEL
LIN {X 0,Y 439.465,Z 263.412,A -85,B 0,C 180,E1 -9061.896,E2 -9061.896} C_VEL
LIN {X 0,Y 440.229,Z 266.73,A -85,B 0,C 180,E1 -9062.653,E2 -9062.653} C_VEL
LIN {X 0,Y 442.895,Z 279.523,A -85,B 0,C 180,E1 -9065.234,E2 -9065.234} C_VEL
LIN {X 0,Y 442.963,Z 283.012,A -85,B 0,C 180,E1 -9065.887,E2 -9065.887} C_VEL
LIN {X 0,Y 442.204,Z 294.955,A -85,B 0,C 180,E1 -9068.008,E2 -9068.008} C_VEL
LIN {X 0,Y 446.763,Z 318.965,A -85,B 0,C 180,E1 -9068.678,E2 -9068.678} C_VEL
LIN {X 0,Y 445.819,Z 409.612,A -85,B 0,C 180,E1 -9070.159,E2 -9070.159} C_VEL
LIN {X 0,Y 445.401,Z 434.069,A -85,B 0,C 180,E1 -9070.589,E2 -9070.589} C_VEL
LIN {X 0,Y 444.885,Z 448.157,A -85,B 0,C 180,E1 -9071.015,E2 -9071.015} C_VEL
LIN {X 0,Y 444.231,Z 461.954,A -85,B 0,C 180,E1 -9071.62,E2 -9071.62} C_VEL
LIN {X 0,Y 443.456,Z 475.275,A -85,B 0,C 180,E1 -9072.4,E2 -9072.4} C_VEL
LIN {X 0,Y 442.7,Z 487.105,A -85,B 0,C 180,E1 -9073.278,E2 -9073.278} C_VEL
LIN {X 0,Y 441.804,Z 498.494,A -85,B 0,C 180,E1 -9074.311,E2 -9074.311} C_VEL
LIN {X 0,Y 441.011,Z 508.96,A -85,B 0,C 180,E1 -9075.464,E2 -9075.464} C_VEL
LIN {X 0,Y 440.289,Z 519.211,A -85,B 0,C 180,E1 -9076.83,E2 -9076.83} C_VEL
LIN {X 0,Y 439.702,Z 527.961,A -85,B 0,C 180,E1 -9078.242,E2 -9078.242} C_VEL
LIN {X 0,Y 439.081,Z 536.184,A -85,B 0,C 180,E1 -9079.859,E2 -9079.859} C_VEL
LIN {X 0,Y 438.779,Z 541.941,A -85,B 0,C 180,E1 -9081.248,E2 -9081.248} C_VEL
LIN {X 0,Y 438.517,Z 546.656,A -85,B 0,C 180,E1 -9082.634,E2 -9082.634} C_VEL
LIN {X 0,Y 438.389,Z 551.543,A -85,B 0,C 180,E1 -9084.48,E2 -9084.48} C_VEL
LIN {X 0,Y 438.25,Z 554.939,A -85,B 0,C 180,E1 -9086.322,E2 -9086.322} C_VEL
LIN {X 0,Y 438.271,Z 556.949,A -85,B 0,C 180,E1 -9088.162,E2 -9088.162} C_VEL
LIN {X 0,Y 438.227,Z 557.614,A -85,B 0,C 180,E1 -9090,E2 -9090} C_VEL
LIN {X 0,Y 438.271,Z 556.948,A -85,B 0,C 180,E1 -9091.838,E2 -9091.838} C_VEL
LIN {X 0,Y 438.25,Z 554.939,A -85,B 0,C 180,E1 -9093.678,E2 -9093.678} C_VEL
LIN {X 0,Y 438.395,Z 551.539,A -85,B 0,C 180,E1 -9095.52,E2 -9095.52} C_VEL
LIN {X 0,Y 438.516,Z 546.645,A -85,B 0,C 180,E1 -9097.366,E2 -9097.366} C_VEL
LIN {X 0,Y 438.888,Z 540.115,A -85,B 0,C 180,E1 -9099.214,E2 -9099.214} C_VEL
LIN {X 0,Y 439.294,Z 532.846,A -85,B 0,C 180,E1 -9100.835,E2 -9100.835} C_VEL
LIN {X 0,Y 439.978,Z 523.845,A -85,B 0,C 180,E1 -9102.453,E2 -9102.453} C_VEL
LIN {X 0,Y 440.637,Z 514.396,A -85,B 0,C 180,E1 -9103.842,E2 -9103.842} C_VEL
LIN {X 0,Y 441.407,Z 503.936,A -85,B 0,C 180,E1 -9105.112,E2 -9105.112} C_VEL
LIN {X 0,Y 442.264,Z 492.393,A -85,B 0,C 180,E1 -9106.265,E2 -9106.265} C_VEL
LIN {X 0,Y 443.109,Z 481.17,A -85,B 0,C 180,E1 -9107.181,E2 -9107.181} C_VEL
LIN {X 0,Y 443.941,Z 468.064,A -85,B 0,C 180,E1 -9108.041,E2 -9108.041} C_VEL
LIN {X 0,Y 444.612,Z 454.452,A -85,B 0,C 180,E1 -9108.728,E2 -9108.728} C_VEL
LIN {X 0,Y 445.221,Z 440.337,A -85,B 0,C 180,E1 -9109.239,E2 -9109.239} C_VEL
LIN {X 0,Y 445.532,Z 426.969,A -85,B 0,C 180,E1 -9109.555,E2 -9109.555} C_VEL
LIN {X 0,Y 446.861,Z 319.869,A -85,B 0,C 180,E1 -9111.297,E2 -9111.297} C_VEL
LIN {X 0,Y 442.448,Z 296.533,A -85,B 0,C 180,E1 -9111.918,E2 -9111.918} C_VEL
LIN {X 0,Y 442.224,Z 294.903,A -85,B 0,C 180,E1 -9111.991,E2 -9111.991} C_VEL
LIN {X 0,Y 443.055,Z 280.561,A -85,B 0,C 180,E1 -9114.556,E2 -9114.556} C_VEL
LIN {X 0,Y 440.512,Z 267.917,A -85,B 0,C 180,E1 -9117.094,E2 -9117.094} C_VEL
LIN {X 0,Y 439.475,Z 263.454,A -85,B 0,C 180,E1 -9118.074,E2 -9118.074} C_VEL
LIN {X 0,Y 439.36,Z 263.363,A -85,B 0,C 180,E1 -9120.788,E2 -9120.788} C_VEL
LIN {X 0,Y 439.385,Z 263.371,A -85,B 0,C 180,E1 -9124.043,E2 -9124.043} C_VEL
LIN {X 0,Y 439.345,Z 263.373,A -85,B 0,C 180,E1 -9126.886,E2 -9126.886} C_VEL
LIN {X 0,Y 439.398,Z 263.376,A -85,B 0,C 180,E1 -9129.849,E2 -9129.849} C_VEL
LIN {X 0,Y 439.384,Z 263.371,A -85,B 0,C 180,E1 -9132.627,E2 -9132.627} C_VEL
LIN {X 0,Y 439.398,Z 263.372,A -85,B 0,C 180,E1 -9135.27,E2 -9135.27} C_VEL
LIN {X 0,Y 439.384,Z 263.373,A -85,B 0,C 180,E1 -9138.743,E2 -9138.743} C_VEL
LIN {X 0,Y 439.38,Z 263.377,A -85,B 0,C 180,E1 -9141.605,E2 -9141.605} C_VEL
LIN {X 0,Y 439.395,Z 263.35,A -85,B 0,C 180,E1 -9144.844,E2 -9144.844} C_VEL
LIN {X 0,Y 439.382,Z 263.372,A -85,B 0,C 180,E1 -9148.14,E2 -9148.14} C_VEL
LIN {X 0,Y 439.419,Z 263.37,A -85,B 0,C 180,E1 -9151.327,E2 -9151.327} C_VEL
LIN {X 0,Y 439.399,Z 263.376,A -85,B 0,C 180,E1 -9154.415,E2 -9154.415} C_VEL
LIN {X 0,Y 439.358,Z 263.376,A -85,B 0,C 180,E1 -9157.424,E2 -9157.424} C_VEL
LIN {X 0,Y 439.434,Z 263.369,A -85,B 0,C 180,E1 -9160.663,E2 -9160.663} C_VEL
LIN {X 0,Y 439.454,Z 263.365,A -85,B 0,C 180,E1 -9164.224,E2 -9164.224} C_VEL
LIN {X 0,Y 439.475,Z 263.362,A -85,B 0,C 180,E1 -9168.001,E2 -9168.001} C_VEL
LIN {X 0,Y 439.54,Z 263.359,A -85,B 0,C 180,E1 -9171.726,E2 -9171.726} C_VEL
LIN {X 0,Y 439.613,Z 263.342,A -85,B 0,C 180,E1 -9174.496,E2 -9174.496} C_VEL
LIN {X 0,Y 439.628,Z 263.345,A -85,B 0,C 180,E1 -9178.168,E2 -9178.168} C_VEL
LIN {X 0,Y 439.755,Z 263.329,A -85,B 0,C 180,E1 -9180,E2 -9180} C_VEL
LIN {X 0,Y 439.649,Z 263.33,A -85,B 0,C 180,E1 -9182.749,E2 -9182.749} C_VEL
LIN {X 0,Y 439.612,Z 263.346,A -85,B 0,C 180,E1 -9186.425,E2 -9186.425} C_VEL
LIN {X 0,Y 439.492,Z 263.356,A -85,B 0,C 180,E1 -9189.202,E2 -9189.202} C_VEL
LIN {X 0,Y 439.461,Z 263.369,A -85,B 0,C 180,E1 -9192.938,E2 -9192.938} C_VEL
LIN {X 0,Y 439.44,Z 263.364,A -85,B 0,C 180,E1 -9196.349,E2 -9196.349} C_VEL
LIN {X 0,Y 439.395,Z 263.37,A -85,B 0,C 180,E1 -9199.627,E2 -9199.627} C_VEL
LIN {X 0,Y 439.358,Z 263.377,A -85,B 0,C 180,E1 -9202.576,E2 -9202.576} C_VEL
LIN {X 0,Y 439.398,Z 263.368,A -85,B 0,C 180,E1 -9205.585,E2 -9205.585} C_VEL
LIN {X 0,Y 439.419,Z 263.374,A -85,B 0,C 180,E1 -9208.673,E2 -9208.673} C_VEL
LIN {X 0,Y 439.369,Z 263.364,A -85,B 0,C 180,E1 -9211.861,E2 -9211.861} C_VEL
LIN {X 0,Y 439.396,Z 263.362,A -85,B 0,C 180,E1 -9215.156,E2 -9215.156} C_VEL
LIN {X 0,Y 439.39,Z 263.38,A -85,B 0,C 180,E1 -9218.594,E2 -9218.594} C_VEL
LIN {X 0,Y 439.394,Z 263.354,A -85,B 0,C 180,E1 -9221.259,E2 -9221.259} C_VEL
LIN {X 0,Y 439.399,Z 263.38,A -85,B 0,C 180,E1 -9224.73,E2 -9224.73} C_VEL
LIN {X 0,Y 439.395,Z 263.359,A -85,B 0,C 180,E1 -9227.797,E2 -9227.797} C_VEL
LIN {X 0,Y 439.434,Z 263.373,A -85,B 0,C 180,E1 -9230.229,E2 -9230.229} C_VEL
LIN {X 0,Y 439.373,Z 263.377,A -85,B 0,C 180,E1 -9233.714,E2 -9233.714} C_VEL
LIN {X 0,Y 439.372,Z 263.381,A -85,B 0,C 180,E1 -9237.055,E2 -9237.055} C_VEL
LIN {X 0,Y 439.382,Z 263.378,A -85,B 0,C 180,E1 -9240.275,E2 -9240.275} C_VEL
LIN {X 0,Y 439.456,Z 263.432,A -85,B 0,C 180,E1 -9243.142,E2 -9243.142} C_VEL
LIN {X 0,Y 441.804,Z 274.595,A -85,B 0,C 180,E1 -9245.57,E2 -9245.57} C_VEL
LIN {X 0,Y 442.774,Z 279.683,A -85,B 0,C 180,E1 -9246.621,E2 -9246.621} C_VEL
LIN {X 0,Y 442.333,Z 287.639,A -85,B 0,C 180,E1 -9248.078,E2 -9248.078} C_VEL
LIN {X 0,Y 446.886,Z 310.046,A -85,B 0,C 180,E1 -9248.715,E2 -9248.715} C_VEL
LIN {X 0,Y 445.72,Z 408.703,A -85,B 0,C 180,E1 -9250.32,E2 -9250.32} C_VEL
LIN {X 0,Y 445.368,Z 427.72,A -85,B 0,C 180,E1 -9250.678,E2 -9250.678} C_VEL
LIN {X 0,Y 445.009,Z 439.021,A -85,B 0,C 180,E1 -9251.021,E2 -9251.021} C_VEL
LIN {X 0,Y 443.437,Z 446.523,A -85,B 0,C 180,E1 -9251.264,E2 -9251.264} C_VEL
LIN {X 0,Y 440.797,Z 453.794,A -85,B 0,C 180,E1 -9251.506,E2 -9251.506} C_VEL
LIN {X 0,Y 437.737,Z 462.71,A -85,B 0,C 180,E1 -9251.892,E2 -9251.892} C_VEL
LIN {X 0,Y 436.837,Z 467.99,A -85,B 0,C 180,E1 -9252.213,E2 -9252.213} C_VEL
LIN {X 0,Y 436.016,Z 480.061,A -85,B 0,C 180,E1 -9253.134,E2 -9253.134} C_VEL
LIN {X 0,Y 435.086,Z 491.272,A -85,B 0,C 180,E1 -9254.182,E2 -9254.182} C_VEL
LIN {X 0,Y 434.189,Z 502.543,A -85,B 0,C 180,E1 -9255.47,E2 -9255.47} C_VEL
LIN {X 0,Y 433.327,Z 512.607,A -85,B 0,C 180,E1 -9256.876,E2 -9256.876} C_VEL
LIN {X 0,Y 432.803,Z 520.961,A -85,B 0,C 180,E1 -9258.289,E2 -9258.289} C_VEL
LIN {X 0,Y 432.179,Z 528.942,A -85,B 0,C 180,E1 -9259.932,E2 -9259.932} C_VEL
LIN {X 0,Y 431.735,Z 535.366,A -85,B 0,C 180,E1 -9261.576,E2 -9261.576} C_VEL
LIN {X 0,Y 431.477,Z 541.206,A -85,B 0,C 180,E1 -9263.507,E2 -9263.507} C_VEL
LIN {X 0,Y 431.281,Z 545.205,A -85,B 0,C 180,E1 -9265.327,E2 -9265.327} C_VEL
LIN {X 0,Y 431.238,Z 547.915,A -85,B 0,C 180,E1 -9267.198,E2 -9267.198} C_VEL
LIN {X 0,Y 431.147,Z 549.275,A -85,B 0,C 180,E1 -9269.066,E2 -9269.066} C_VEL
LIN {X 0,Y 431.147,Z 549.313,A -85,B 0,C 180,E1 -9270.934,E2 -9270.934} C_VEL
LIN {X 0,Y 431.237,Z 548.023,A -85,B 0,C 180,E1 -9272.802,E2 -9272.802} C_VEL
LIN {X 0,Y 431.281,Z 545.378,A -85,B 0,C 180,E1 -9274.673,E2 -9274.673} C_VEL
LIN {X 0,Y 431.486,Z 541.309,A -85,B 0,C 180,E1 -9276.547,E2 -9276.547} C_VEL
LIN {X 0,Y 431.729,Z 535.688,A -85,B 0,C 180,E1 -9278.424,E2 -9278.424} C_VEL
LIN {X 0,Y 432.165,Z 529.341,A -85,B 0,C 180,E1 -9280.068,E2 -9280.068} C_VEL
LIN {X 0,Y 432.75,Z 521.449,A -85,B 0,C 180,E1 -9281.712,E2 -9281.712} C_VEL
LIN {X 0,Y 433.318,Z 513.194,A -85,B 0,C 180,E1 -9283.124,E2 -9283.124} C_VEL
LIN {X 0,Y 434.116,Z 503.246,A -85,B 0,C 180,E1 -9284.532,E2 -9284.532} C_VEL
LIN {X 0,Y 435.008,Z 492.175,A -85,B 0,C 180,E1 -9285.821,E2 -9285.821} C_VEL
LIN {X 0,Y 435.905,Z 481.151,A -85,B 0,C 180,E1 -9286.87,E2 -9286.87} C_VEL
LIN {X 0,Y 436.841,Z 468.032,A -85,B 0,C 180,E1 -9287.879,E2 -9287.879} C_VEL
LIN {X 0,Y 437.602,Z 454.881,A -85,B 0,C 180,E1 -9288.672,E2 -9288.672} C_VEL
LIN {X 0,Y 438.27,Z 440.707,A -85,B 0,C 180,E1 -9289.313,E2 -9289.313} C_VEL
LIN {X 0,Y 438.789,Z 426.813,A -85,B 0,C 180,E1 -9289.746,E2 -9289.746} C_VEL
LIN {X 0,Y 439.167,Z 402.682,A -85,B 0,C 180,E1 -9290.185,E2 -9290.185} C_VEL
LIN {X 0,Y 440.332,Z 311.667,A -85,B 0,C 180,E1 -9291.686,E2 -9291.686} C_VEL
LIN {X 0,Y 435.782,Z 289.139,A -85,B 0,C 180,E1 -9292.318,E2 -9292.318} C_VEL
LIN {X 0,Y 435.498,Z 287.394,A -85,B 0,C 180,E1 -9292.41,E2 -9292.41} C_VEL
LIN {X 0,Y 435.867,Z 282.148,A -85,B 0,C 180,E1 -9293.394,E2 -9293.394} C_VEL
LIN {X 0,Y 434.984,Z 276.415,A -85,B 0,C 180,E1 -9294.584,E2 -9294.584} C_VEL
LIN {X 0,Y 432.438,Z 264.466,A -85,B 0,C 180,E1 -9297.199,E2 -9297.199} C_VEL
LIN {X 0,Y 432.342,Z 264.244,A -85,B 0,C 180,E1 -9299.187,E2 -9299.187} C_VEL
LIN {X 0,Y 432.322,Z 264.258,A -85,B 0,C 180,E1 -9302.442,E2 -9302.442} C_VEL
LIN {X 0,Y 432.343,Z 264.259,A -85,B 0,C 180,E1 -9305.631,E2 -9305.631} C_VEL
LIN {X 0,Y 432.352,Z 264.254,A -85,B 0,C 180,E1 -9309.341,E2 -9309.341} C_VEL
LIN {X 0,Y 432.332,Z 264.243,A -85,B 0,C 180,E1 -9311.796,E2 -9311.796} C_VEL
LIN {X 0,Y 432.337,Z 264.253,A -85,B 0,C 180,E1 -9314.346,E2 -9314.346} C_VEL
LIN {X 0,Y 432.316,Z 264.251,A -85,B 0,C 180,E1 -9317.015,E2 -9317.015} C_VEL
LIN {X 0,Y 432.351,Z 264.244,A -85,B 0,C 180,E1 -9319.816,E2 -9319.816} C_VEL
LIN {X 0,Y 432.312,Z 264.264,A -85,B 0,C 180,E1 -9323.022,E2 -9323.022} C_VEL
LIN {X 0,Y 432.354,Z 264.229,A -85,B 0,C 180,E1 -9325.996,E2 -9325.996} C_VEL
LIN {X 0,Y 432.389,Z 264.247,A -85,B 0,C 180,E1 -9329.743,E2 -9329.743} C_VEL
LIN {X 0,Y 432.393,Z 264.241,A -85,B 0,C 180,E1 -9333.372,E2 -9333.372} C_VEL
LIN {X 0,Y 432.364,Z 264.25,A -85,B 0,C 180,E1 -9336.023,E2 -9336.023} C_VEL
LIN {X 0,Y 432.342,Z 264.248,A -85,B 0,C 180,E1 -9339.046,E2 -9339.046} C_VEL
LIN {X 0,Y 432.37,Z 264.249,A -85,B 0,C 180,E1 -9342.011,E2 -9342.011} C_VEL
LIN {X 0,Y 432.387,Z 264.241,A -85,B 0,C 180,E1 -9344.926,E2 -9344.926} C_VEL
LIN {X 0,Y 432.451,Z 264.238,A -85,B 0,C 180,E1 -9347.803,E2 -9347.803} C_VEL
LIN {X 0,Y 432.483,Z 264.226,A -85,B 0,C 180,E1 -9351.59,E2 -9351.59} C_VEL
LIN {X 0,Y 432.591,Z 264.225,A -85,B 0,C 180,E1 -9354.406,E2 -9354.406} C_VEL
LIN {X 0,Y 432.597,Z 264.21,A -85,B 0,C 180,E1 -9358.138,E2 -9358.138} C_VEL
LIN {X 0,Y 432.726,Z 264.204,A -85,B 0,C 180,E1 -9360,E2 -9360} C_VEL
LIN {X 0,Y 432.597,Z 264.215,A -85,B 0,C 180,E1 -9362.794,E2 -9362.794} C_VEL
LIN {X 0,Y 432.564,Z 264.23,A -85,B 0,C 180,E1 -9366.53,E2 -9366.53} C_VEL
LIN {X 0,Y 432.434,Z 264.235,A -85,B 0,C 180,E1 -9369.353,E2 -9369.353} C_VEL
LIN {X 0,Y 432.422,Z 264.244,A -85,B 0,C 180,E1 -9372.804,E2 -9372.804} C_VEL
LIN {X 0,Y 432.404,Z 264.239,A -85,B 0,C 180,E1 -9376.479,E2 -9376.479} C_VEL
LIN {X 0,Y 432.331,Z 264.259,A -85,B 0,C 180,E1 -9379.961,E2 -9379.961} C_VEL
LIN {X 0,Y 432.311,Z 264.252,A -85,B 0,C 180,E1 -9382.965,E2 -9382.965} C_VEL
LIN {X 0,Y 432.357,Z 264.252,A -85,B 0,C 180,E1 -9386.033,E2 -9386.033} C_VEL
LIN {X 0,Y 432.345,Z 264.252,A -85,B 0,C 180,E1 -9389.187,E2 -9389.187} C_VEL
LIN {X 0,Y 432.325,Z 264.244,A -85,B 0,C 180,E1 -9392.295,E2 -9392.295} C_VEL
LIN {X 0,Y 432.334,Z 264.228,A -85,B 0,C 180,E1 -9394.678,E2 -9394.678} C_VEL
LIN {X 0,Y 432.341,Z 264.257,A -85,B 0,C 180,E1 -9398.149,E2 -9398.149} C_VEL
LIN {X 0,Y 432.328,Z 264.256,A -85,B 0,C 180,E1 -9401.603,E2 -9401.603} C_VEL
LIN {X 0,Y 432.329,Z 264.254,A -85,B 0,C 180,E1 -9404.348,E2 -9404.348} C_VEL
LIN {X 0,Y 432.362,Z 264.25,A -85,B 0,C 180,E1 -9407.01,E2 -9407.01} C_VEL
LIN {X 0,Y 432.354,Z 264.25,A -85,B 0,C 180,E1 -9409.818,E2 -9409.818} C_VEL
LIN {X 0,Y 432.312,Z 264.248,A -85,B 0,C 180,E1 -9413.024,E2 -9413.024} C_VEL
LIN {X 0,Y 432.357,Z 264.246,A -85,B 0,C 180,E1 -9415.997,E2 -9415.997} C_VEL
LIN {X 0,Y 432.345,Z 264.231,A -85,B 0,C 180,E1 -9419.49,E2 -9419.49} C_VEL
LIN {X 0,Y 432.415,Z 264.371,A -85,B 0,C 180,E1 -9421.62,E2 -9421.62} C_VEL
LIN {X 0,Y 434.773,Z 274.881,A -85,B 0,C 180,E1 -9423.866,E2 -9423.866} C_VEL
LIN {X 0,Y 436.214,Z 282.95,A -85,B 0,C 180,E1 -9425.49,E2 -9425.49} C_VEL
LIN {X 0,Y 435.372,Z 294.892,A -85,B 0,C 180,E1 -9427.644,E2 -9427.644} C_VEL
LIN {X 0,Y 439.869,Z 318.209,A -85,B 0,C 180,E1 -9428.315,E2 -9428.315} C_VEL
LIN {X 0,Y 440.242,Z 322.253,A -85,B 0,C 180,E1 -9428.404,E2 -9428.404} C_VEL
LIN {X 0,Y 438.9,Z 425.636,A -85,B 0,C 180,E1 -9430.107,E2 -9430.107} C_VEL
LIN {X 0,Y 438.458,Z 440.423,A -85,B 0,C 180,E1 -9430.452,E2 -9430.452} C_VEL
LIN {X 0,Y 437.884,Z 454.5,A -85,B 0,C 180,E1 -9430.974,E2 -9430.974} C_VEL
LIN {X 0,Y 437.149,Z 468.55,A -85,B 0,C 180,E1 -9431.698,E2 -9431.698} C_VEL
LIN {X 0,Y 436.319,Z 481.158,A -85,B 0,C 180,E1 -9432.543,E2 -9432.543} C_VEL
LIN {X 0,Y 435.322,Z 493.665,A -85,B 0,C 180,E1 -9433.589,E2 -9433.589} C_VEL
LIN {X 0,Y 434.487,Z 504.974,A -85,B 0,C 180,E1 -9434.761,E2 -9434.761} C_VEL
LIN {X 0,Y 433.682,Z 514.359,A -85,B 0,C 180,E1 -9435.932,E2 -9435.932} C_VEL
LIN {X 0,Y 432.998,Z 523.802,A -85,B 0,C 180,E1 -9437.343,E2 -9437.343} C_VEL
LIN {X 0,Y 432.294,Z 532.796,A -85,B 0,C 180,E1 -9438.988,E2 -9438.988} C_VEL
LIN {X 0,Y 431.809,Z 540.061,A -85,B 0,C 180,E1 -9440.633,E2 -9440.633} C_VEL
LIN {X 0,Y 431.448,Z 546.591,A -85,B 0,C 180,E1 -9442.512,E2 -9442.512} C_VEL
LIN {X 0,Y 431.292,Z 551.477,A -85,B 0,C 180,E1 -9444.389,E2 -9444.389} C_VEL
LIN {X 0,Y 431.159,Z 554.873,A -85,B 0,C 180,E1 -9446.262,E2 -9446.262} C_VEL
LIN {X 0,Y 431.194,Z 556.882,A -85,B 0,C 180,E1 -9448.132,E2 -9448.132} C_VEL
LIN {X 0,Y 431.142,Z 557.547,A -85,B 0,C 180,E1 -9450,E2 -9450} C_VEL
LIN {X 0,Y 431.194,Z 556.881,A -85,B 0,C 180,E1 -9451.868,E2 -9451.868} C_VEL
LIN {X 0,Y 431.159,Z 554.872,A -85,B 0,C 180,E1 -9453.738,E2 -9453.738} C_VEL
LIN {X 0,Y 431.297,Z 551.472,A -85,B 0,C 180,E1 -9455.611,E2 -9455.611} C_VEL
LIN {X 0,Y 431.447,Z 546.578,A -85,B 0,C 180,E1 -9457.488,E2 -9457.488} C_VEL
LIN {X 0,Y 431.825,Z 540.046,A -85,B 0,C 180,E1 -9459.366,E2 -9459.366} C_VEL
LIN {X 0,Y 432.294,Z 532.778,A -85,B 0,C 180,E1 -9461.012,E2 -9461.012} C_VEL
LIN {X 0,Y 432.915,Z 525.16,A -85,B 0,C 180,E1 -9462.421,E2 -9462.421} C_VEL
LIN {X 0,Y 433.568,Z 516.182,A -85,B 0,C 180,E1 -9463.809,E2 -9463.809} C_VEL
LIN {X 0,Y 434.28,Z 506.906,A -85,B 0,C 180,E1 -9465.006,E2 -9465.006} C_VEL
LIN {X 0,Y 435.138,Z 496.035,A -85,B 0,C 180,E1 -9466.177,E2 -9466.177} C_VEL
LIN {X 0,Y 436.12,Z 484.135,A -85,B 0,C 180,E1 -9467.224,E2 -9467.224} C_VEL
LIN {X 0,Y 436.922,Z 471.793,A -85,B 0,C 180,E1 -9468.102,E2 -9468.102} C_VEL
LIN {X 0,Y 437.708,Z 458.264,A -85,B 0,C 180,E1 -9468.852,E2 -9468.852} C_VEL
LIN {X 0,Y 438.316,Z 444.834,A -85,B 0,C 180,E1 -9469.402,E2 -9469.402} C_VEL
LIN {X 0,Y 438.741,Z 431.4,A -85,B 0,C 180,E1 -9469.779,E2 -9469.779} C_VEL
LIN {X 0,Y 440.084,Z 333.369,A -85,B 0,C 180,E1 -9471.408,E2 -9471.408} C_VEL
LIN {X 0,Y 440.136,Z 319.746,A -85,B 0,C 180,E1 -9471.639,E2 -9471.639} C_VEL
LIN {X 0,Y 435.416,Z 295.183,A -85,B 0,C 180,E1 -9472.327,E2 -9472.327} C_VEL
LIN {X 0,Y 435.515,Z 292.296,A -85,B 0,C 180,E1 -9472.786,E2 -9472.786} C_VEL
LIN {X 0,Y 436.184,Z 282.907,A -85,B 0,C 180,E1 -9474.512,E2 -9474.512} C_VEL
LIN {X 0,Y 434.491,Z 273.497,A -85,B 0,C 180,E1 -9476.411,E2 -9476.411} C_VEL
LIN {X 0,Y 432.415,Z 264.352,A -85,B 0,C 180,E1 -9478.38,E2 -9478.38} C_VEL
LIN {X 0,Y 432.32,Z 264.251,A -85,B 0,C 180,E1 -9481.345,E2 -9481.345} C_VEL
LIN {X 0,Y 432.337,Z 264.256,A -85,B 0,C 180,E1 -9484.676,E2 -9484.676} C_VEL
LIN {X 0,Y 432.334,Z 264.251,A -85,B 0,C 180,E1 -9488.149,E2 -9488.149} C_VEL
LIN {X 0,Y 432.331,Z 264.24,A -85,B 0,C 180,E1 -9491.602,E2 -9491.602} C_VEL
LIN {X 0,Y 432.338,Z 264.26,A -85,B 0,C 180,E1 -9494.346,E2 -9494.346} C_VEL
LIN {X 0,Y 432.316,Z 264.257,A -85,B 0,C 180,E1 -9497.015,E2 -9497.015} C_VEL
LIN {X 0,Y 432.336,Z 264.25,A -85,B 0,C 180,E1 -9499.819,E2 -9499.819} C_VEL
LIN {X 0,Y 432.31,Z 264.251,A -85,B 0,C 180,E1 -9503.022,E2 -9503.022} C_VEL
LIN {X 0,Y 432.354,Z 264.226,A -85,B 0,C 180,E1 -9505.996,E2 -9505.996} C_VEL
LIN {X 0,Y 432.389,Z 264.249,A -85,B 0,C 180,E1 -9509.744,E2 -9509.744} C_VEL
LIN {X 0,Y 432.394,Z 264.241,A -85,B 0,C 180,E1 -9513.372,E2 -9513.372} C_VEL
LIN {X 0,Y 432.364,Z 264.252,A -85,B 0,C 180,E1 -9516.023,E2 -9516.023} C_VEL
LIN {X 0,Y 432.342,Z 264.249,A -85,B 0,C 180,E1 -9519.046,E2 -9519.046} C_VEL
LIN {X 0,Y 432.371,Z 264.248,A -85,B 0,C 180,E1 -9522.011,E2 -9522.011} C_VEL
LIN {X 0,Y 432.387,Z 264.243,A -85,B 0,C 180,E1 -9524.926,E2 -9524.926} C_VEL
LIN {X 0,Y 432.451,Z 264.24,A -85,B 0,C 180,E1 -9527.803,E2 -9527.803} C_VEL
LIN {X 0,Y 432.484,Z 264.236,A -85,B 0,C 180,E1 -9531.59,E2 -9531.59} C_VEL
LIN {X 0,Y 432.59,Z 264.217,A -85,B 0,C 180,E1 -9534.406,E2 -9534.406} C_VEL
LIN {X 0,Y 432.598,Z 264.221,A -85,B 0,C 180,E1 -9538.138,E2 -9538.138} C_VEL
LIN {X 0,Y 432.725,Z 264.204,A -85,B 0,C 180,E1 -9540,E2 -9540} C_VEL
LIN {X 0,Y 432.598,Z 264.208,A -85,B 0,C 180,E1 -9542.794,E2 -9542.794} C_VEL
LIN {X 0,Y 432.566,Z 264.224,A -85,B 0,C 180,E1 -9546.531,E2 -9546.531} C_VEL
LIN {X 0,Y 432.435,Z 264.235,A -85,B 0,C 180,E1 -9549.353,E2 -9549.353} C_VEL
LIN {X 0,Y 432.424,Z 264.244,A -85,B 0,C 180,E1 -9552.804,E2 -9552.804} C_VEL
LIN {X 0,Y 432.405,Z 264.241,A -85,B 0,C 180,E1 -9556.479,E2 -9556.479} C_VEL
LIN {X 0,Y 432.331,Z 264.248,A -85,B 0,C 180,E1 -9559.961,E2 -9559.961} C_VEL
LIN {X 0,Y 432.312,Z 264.259,A -85,B 0,C 180,E1 -9562.965,E2 -9562.965} C_VEL
LIN {X 0,Y 432.358,Z 264.243,A -85,B 0,C 180,E1 -9566.033,E2 -9566.033} C_VEL
LIN {X 0,Y 432.347,Z 264.255,A -85,B 0,C 180,E1 -9569.187,E2 -9569.187} C_VEL
LIN {X 0,Y 432.32,Z 264.239,A -85,B 0,C 180,E1 -9572.294,E2 -9572.294} C_VEL
LIN {X 0,Y 432.336,Z 264.232,A -85,B 0,C 180,E1 -9574.678,E2 -9574.678} C_VEL
LIN {X 0,Y 432.346,Z 264.254,A -85,B 0,C 180,E1 -9578.149,E2 -9578.149} C_VEL
LIN {X 0,Y 432.363,Z 264.229,A -85,B 0,C 180,E1 -9581.608,E2 -9581.608} C_VEL
LIN {X 0,Y 432.33,Z 264.255,A -85,B 0,C 180,E1 -9584.348,E2 -9584.348} C_VEL
LIN {X 0,Y 432.322,Z 264.243,A -85,B 0,C 180,E1 -9587.016,E2 -9587.016} C_VEL
LIN {X 0,Y 432.339,Z 264.254,A -85,B 0,C 180,E1 -9589.82,E2 -9589.82} C_VEL
LIN {X 0,Y 432.306,Z 264.256,A -85,B 0,C 180,E1 -9593.023,E2 -9593.023} C_VEL
LIN {X 0,Y 432.358,Z 264.247,A -85,B 0,C 180,E1 -9595.997,E2 -9595.997} C_VEL
LIN {X 0,Y 432.347,Z 264.255,A -85,B 0,C 180,E1 -9599.49,E2 -9599.49} C_VEL
LIN {X 0,Y 432.441,Z 264.366,A -85,B 0,C 180,E1 -9602.867,E2 -9602.867} C_VEL
LIN {X 0,Y 435.153,Z 277.208,A -85,B 0,C 180,E1 -9605.68,E2 -9605.68} C_VEL
LIN {X 0,Y 435.841,Z 282.652,A -85,B 0,C 180,E1 -9606.8,E2 -9606.8} C_VEL
LIN {X 0,Y 435.532,Z 287.773,A -85,B 0,C 180,E1 -9607.722,E2 -9607.722} C_VEL
LIN {X 0,Y 440.312,Z 311.638,A -85,B 0,C 180,E1 -9608.407,E2 -9608.407} C_VEL
LIN {X 0,Y 439.077,Z 407.827,A -85,B 0,C 180,E1 -9609.993,E2 -9609.993} C_VEL
LIN {X 0,Y 438.687,Z 427.804,A -85,B 0,C 180,E1 -9610.371,E2 -9610.371} C_VEL
LIN {X 0,Y 438.139,Z 442.119,A -85,B 0,C 180,E1 -9610.833,E2 -9610.833} C_VEL
LIN {X 0,Y 437.581,Z 455.591,A -85,B 0,C 180,E1 -9611.46,E2 -9611.46} C_VEL
LIN {X 0,Y 436.837,Z 467.99,A -85,B 0,C 180,E1 -9612.213,E2 -9612.213} C_VEL
LIN {X 0,Y 435.862,Z 473.203,A -85,B 0,C 180,E1 -9612.557,E2 -9612.557} C_VEL
LIN {X 0,Y 432.48,Z 481.525,A -85,B 0,C 180,E1 -9613.116,E2 -9613.116} C_VEL
LIN {X 0,Y 429.067,Z 489.481,A -85,B 0,C 180,E1 -9613.757,E2 -9613.757} C_VEL
LIN {X 0,Y 428.05,Z 494.114,A -85,B 0,C 180,E1 -9614.225,E2 -9614.225} C_VEL
LIN {X 0,Y 427.108,Z 504.393,A -85,B 0,C 180,E1 -9615.467,E2 -9615.467} C_VEL
LIN {X 0,Y 426.316,Z 514.159,A -85,B 0,C 180,E1 -9616.899,E2 -9616.899} C_VEL
LIN {X 0,Y 425.705,Z 522.259,A -85,B 0,C 180,E1 -9618.332,E2 -9618.332} C_VEL
LIN {X 0,Y 425.062,Z 530.016,A -85,B 0,C 180,E1 -9620.003,E2 -9620.003} C_VEL
LIN {X 0,Y 424.68,Z 535.435,A -85,B 0,C 180,E1 -9621.435,E2 -9621.435} C_VEL
LIN {X 0,Y 424.399,Z 541.131,A -85,B 0,C 180,E1 -9623.343,E2 -9623.343} C_VEL
LIN {X 0,Y 424.212,Z 545.272,A -85,B 0,C 180,E1 -9625.248,E2 -9625.248} C_VEL
LIN {X 0,Y 424.135,Z 547.982,A -85,B 0,C 180,E1 -9627.151,E2 -9627.151} C_VEL
LIN {X 0,Y 424.068,Z 549.342,A -85,B 0,C 180,E1 -9629.05,E2 -9629.05} C_VEL
LIN {X 0,Y 424.068,Z 549.379,A -85,B 0,C 180,E1 -9630.95,E2 -9630.95} C_VEL
LIN {X 0,Y 424.134,Z 548.089,A -85,B 0,C 180,E1 -9632.849,E2 -9632.849} C_VEL
LIN {X 0,Y 424.212,Z 545.444,A -85,B 0,C 180,E1 -9634.751,E2 -9634.751} C_VEL
LIN {X 0,Y 424.401,Z 541.375,A -85,B 0,C 180,E1 -9636.656,E2 -9636.656} C_VEL
LIN {X 0,Y 424.674,Z 535.754,A -85,B 0,C 180,E1 -9638.565,E2 -9638.565} C_VEL
LIN {X 0,Y 425.153,Z 529.406,A -85,B 0,C 180,E1 -9640.236,E2 -9640.236} C_VEL
LIN {X 0,Y 425.771,Z 521.513,A -85,B 0,C 180,E1 -9641.907,E2 -9641.907} C_VEL
LIN {X 0,Y 426.367,Z 513.258,A -85,B 0,C 180,E1 -9643.342,E2 -9643.342} C_VEL
LIN {X 0,Y 427.21,Z 503.31,A -85,B 0,C 180,E1 -9644.773,E2 -9644.773} C_VEL
LIN {X 0,Y 428.166,Z 492.237,A -85,B 0,C 180,E1 -9646.08,E2 -9646.08} C_VEL
LIN {X 0,Y 429.105,Z 481.213,A -85,B 0,C 180,E1 -9647.146,E2 -9647.146} C_VEL
LIN {X 0,Y 430.088,Z 468.177,A -85,B 0,C 180,E1 -9648.163,E2 -9648.163} C_VEL
LIN {X 0,Y 430.883,Z 454.848,A -85,B 0,C 180,E1 -9648.98,E2 -9648.98} C_VEL
LIN {X 0,Y 431.568,Z 440.762,A -85,B 0,C 180,E1 -9649.625,E2 -9649.625} C_VEL
LIN {X 0,Y 432.113,Z 426.862,A -85,B 0,C 180,E1 -9650.064,E2 -9650.064} C_VEL
LIN {X 0,Y 432.53,Z 402.722,A -85,B 0,C 180,E1 -9650.509,E2 -9650.509} C_VEL
LIN {X 0,Y 433.683,Z 311.8,A -85,B 0,C 180,E1 -9652.035,E2 -9652.035} C_VEL
LIN {X 0,Y 428.672,Z 287.684,A -85,B 0,C 180,E1 -9652.764,E2 -9652.764} C_VEL
LIN {X 0,Y 428.93,Z 282.558,A -85,B 0,C 180,E1 -9653.726,E2 -9653.726} C_VEL
LIN {X 0,Y 426.415,Z 270.121,A -85,B 0,C 180,E1 -9656.423,E2 -9656.423} C_VEL
LIN {X 0,Y 425.384,Z 265.251,A -85,B 0,C 180,E1 -9657.554,E2 -9657.554} C_VEL
LIN {X 0,Y 425.287,Z 265.133,A -85,B 0,C 180,E1 -9660.815,E2 -9660.815} C_VEL
LIN {X 0,Y 425.31,Z 265.125,A -85,B 0,C 180,E1 -9664.287,E2 -9664.287} C_VEL
LIN {X 0,Y 425.278,Z 265.128,A -85,B 0,C 180,E1 -9667.693,E2 -9667.693} C_VEL
LIN {X 0,Y 425.282,Z 265.134,A -85,B 0,C 180,E1 -9670.52,E2 -9670.52} C_VEL
LIN {X 0,Y 425.265,Z 265.135,A -85,B 0,C 180,E1 -9673.954,E2 -9673.954} C_VEL
LIN {X 0,Y 425.278,Z 265.12,A -85,B 0,C 180,E1 -9677.347,E2 -9677.347} C_VEL
LIN {X 0,Y 425.304,Z 265.121,A -85,B 0,C 180,E1 -9679.875,E2 -9679.875} C_VEL
LIN {X 0,Y 425.281,Z 265.135,A -85,B 0,C 180,E1 -9682.486,E2 -9682.486} C_VEL
LIN {X 0,Y 425.302,Z 265.107,A -85,B 0,C 180,E1 -9685.817,E2 -9685.817} C_VEL
LIN {X 0,Y 425.294,Z 265.126,A -85,B 0,C 180,E1 -9689.236,E2 -9689.236} C_VEL
LIN {X 0,Y 425.343,Z 265.126,A -85,B 0,C 180,E1 -9692.442,E2 -9692.442} C_VEL
LIN {X 0,Y 425.344,Z 265.126,A -85,B 0,C 180,E1 -9695.602,E2 -9695.602} C_VEL
LIN {X 0,Y 425.285,Z 265.129,A -85,B 0,C 180,E1 -9698.681,E2 -9698.681} C_VEL
LIN {X 0,Y 425.325,Z 265.127,A -85,B 0,C 180,E1 -9701.702,E2 -9701.702} C_VEL
LIN {X 0,Y 425.34,Z 265.12,A -85,B 0,C 180,E1 -9704.67,E2 -9704.67} C_VEL
LIN {X 0,Y 425.404,Z 265.117,A -85,B 0,C 180,E1 -9707.598,E2 -9707.598} C_VEL
LIN {X 0,Y 425.434,Z 265.104,A -85,B 0,C 180,E1 -9711.45,E2 -9711.45} C_VEL
LIN {X 0,Y 425.548,Z 265.102,A -85,B 0,C 180,E1 -9714.313,E2 -9714.313} C_VEL
LIN {X 0,Y 425.567,Z 265.085,A -85,B 0,C 180,E1 -9718.107,E2 -9718.107} C_VEL
LIN {X 0,Y 425.696,Z 265.08,A -85,B 0,C 180,E1 -9720,E2 -9720} C_VEL
LIN {X 0,Y 425.549,Z 265.093,A -85,B 0,C 180,E1 -9722.84,E2 -9722.84} C_VEL
LIN {X 0,Y 425.522,Z 265.106,A -85,B 0,C 180,E1 -9726.639,E2 -9726.639} C_VEL
LIN {X 0,Y 425.393,Z 265.112,A -85,B 0,C 180,E1 -9729.509,E2 -9729.509} C_VEL
LIN {X 0,Y 425.385,Z 265.12,A -85,B 0,C 180,E1 -9732.904,E2 -9732.904} C_VEL
LIN {X 0,Y 425.353,Z 265.117,A -85,B 0,C 180,E1 -9736.605,E2 -9736.605} C_VEL
LIN {X 0,Y 425.32,Z 265.129,A -85,B 0,C 180,E1 -9739.636,E2 -9739.636} C_VEL
LIN {X 0,Y 425.299,Z 265.126,A -85,B 0,C 180,E1 -9743.366,E2 -9743.366} C_VEL
LIN {X 0,Y 425.341,Z 265.118,A -85,B 0,C 180,E1 -9746.845,E2 -9746.845} C_VEL
LIN {X 0,Y 425.311,Z 265.132,A -85,B 0,C 180,E1 -9749.718,E2 -9749.718} C_VEL
LIN {X 0,Y 425.278,Z 265.119,A -85,B 0,C 180,E1 -9753.048,E2 -9753.048} C_VEL
LIN {X 0,Y 425.278,Z 265.117,A -85,B 0,C 180,E1 -9755.93,E2 -9755.93} C_VEL
LIN {X 0,Y 425.298,Z 265.131,A -85,B 0,C 180,E1 -9759.045,E2 -9759.045} C_VEL
LIN {X 0,Y 425.27,Z 265.134,A -85,B 0,C 180,E1 -9762.654,E2 -9762.654} C_VEL
LIN {X 0,Y 425.315,Z 265.129,A -85,B 0,C 180,E1 -9766.052,E2 -9766.052} C_VEL
LIN {X 0,Y 425.306,Z 265.115,A -85,B 0,C 180,E1 -9768.626,E2 -9768.626} C_VEL
LIN {X 0,Y 425.32,Z 265.131,A -85,B 0,C 180,E1 -9771.105,E2 -9771.105} C_VEL
LIN {X 0,Y 425.297,Z 265.133,A -85,B 0,C 180,E1 -9774.665,E2 -9774.665} C_VEL
LIN {X 0,Y 425.263,Z 265.137,A -85,B 0,C 180,E1 -9778.074,E2 -9778.074} C_VEL
LIN {X 0,Y 425.363,Z 265.263,A -85,B 0,C 180,E1 -9781.301,E2 -9781.301} C_VEL
LIN {X 0,Y 427.822,Z 276.162,A -85,B 0,C 180,E1 -9783.671,E2 -9783.671} C_VEL
LIN {X 0,Y 429.332,Z 284.227,A -85,B 0,C 180,E1 -9785.329,E2 -9785.329} C_VEL
LIN {X 0,Y 428.585,Z 294.827,A -85,B 0,C 180,E1 -9787.271,E2 -9787.271} C_VEL
LIN {X 0,Y 433.586,Z 321.055,A -85,B 0,C 180,E1 -9788.035,E2 -9788.035} C_VEL
LIN {X 0,Y 432.296,Z 422.039,A -85,B 0,C 180,E1 -9789.728,E2 -9789.728} C_VEL
LIN {X 0,Y 431.945,Z 437.381,A -85,B 0,C 180,E1 -9790.052,E2 -9790.052} C_VEL
LIN {X 0,Y 431.267,Z 451.822,A -85,B 0,C 180,E1 -9790.546,E2 -9790.546} C_VEL
LIN {X 0,Y 430.586,Z 465.194,A -85,B 0,C 180,E1 -9791.204,E2 -9791.204} C_VEL
LIN {X 0,Y 429.718,Z 477.93,A -85,B 0,C 180,E1 -9792.02,E2 -9792.02} C_VEL
LIN {X 0,Y 428.828,Z 489.723,A -85,B 0,C 180,E1 -9792.966,E2 -9792.966} C_VEL
LIN {X 0,Y 427.828,Z 501.703,A -85,B 0,C 180,E1 -9794.152,E2 -9794.152} C_VEL
LIN {X 0,Y 426.9,Z 512.51,A -85,B 0,C 180,E1 -9795.46,E2 -9795.46} C_VEL
LIN {X 0,Y 426.158,Z 521.814,A -85,B 0,C 180,E1 -9796.823,E2 -9796.823} C_VEL
LIN {X 0,Y 425.528,Z 530.329,A -85,B 0,C 180,E1 -9798.328,E2 -9798.328} C_VEL
LIN {X 0,Y 424.914,Z 538.072,A -85,B 0,C 180,E1 -9799.999,E2 -9799.999} C_VEL
LIN {X 0,Y 424.577,Z 543.477,A -85,B 0,C 180,E1 -9801.433,E2 -9801.433} C_VEL
LIN {X 0,Y 424.298,Z 549.163,A -85,B 0,C 180,E1 -9803.342,E2 -9803.342} C_VEL
LIN {X 0,Y 424.178,Z 553.288,A -85,B 0,C 180,E1 -9805.248,E2 -9805.248} C_VEL
LIN {X 0,Y 424.081,Z 555.981,A -85,B 0,C 180,E1 -9807.15,E2 -9807.15} C_VEL
LIN {X 0,Y 424.067,Z 557.315,A -85,B 0,C 180,E1 -9809.05,E2 -9809.05} C_VEL
LIN {X 0,Y 424.067,Z 557.314,A -85,B 0,C 180,E1 -9810.95,E2 -9810.95} C_VEL
LIN {X 0,Y 424.082,Z 555.979,A -85,B 0,C 180,E1 -9812.85,E2 -9812.85} C_VEL
LIN {X 0,Y 424.18,Z 553.284,A -85,B 0,C 180,E1 -9814.752,E2 -9814.752} C_VEL
LIN {X 0,Y 424.297,Z 549.152,A -85,B 0,C 180,E1 -9816.658,E2 -9816.658} C_VEL
LIN {X 0,Y 424.579,Z 543.46,A -85,B 0,C 180,E1 -9818.567,E2 -9818.567} C_VEL
LIN {X 0,Y 424.951,Z 537.043,A -85,B 0,C 180,E1 -9820.241,E2 -9820.241} C_VEL
LIN {X 0,Y 425.624,Z 529.072,A -85,B 0,C 180,E1 -9821.911,E2 -9821.911} C_VEL
LIN {X 0,Y 426.248,Z 520.431,A -85,B 0,C 180,E1 -9823.395,E2 -9823.395} C_VEL
LIN {X 0,Y 427.055,Z 510.69,A -85,B 0,C 180,E1 -9824.778,E2 -9824.778} C_VEL
LIN {X 0,Y 428.021,Z 499.488,A -85,B 0,C 180,E1 -9826.086,E2 -9826.086} C_VEL
LIN {X 0,Y 428.982,Z 488.344,A -85,B 0,C 180,E1 -9827.151,E2 -9827.151} C_VEL
LIN {X 0,Y 429.898,Z 476.205,A -85,B 0,C 180,E1 -9828.096,E2 -9828.096} C_VEL
LIN {X 0,Y 430.693,Z 464.309,A -85,B 0,C 180,E1 -9828.837,E2 -9828.837} C_VEL
LIN {X 0,Y 431.372,Z 450.17,A -85,B 0,C 180,E1 -9829.511,E2 -9829.511} C_VEL
LIN {X 0,Y 431.952,Z 436.017,A -85,B 0,C 180,E1 -9829.979,E2 -9829.979} C_VEL
LIN {X 0,Y 432.375,Z 418.118,A -85,B 0,C 180,E1 -9830.33,E2 -9830.33} C_VEL
LIN {X 0,Y 433.579,Z 320.921,A -85,B 0,C 180,E1 -9831.961,E2 -9831.961} C_VEL
LIN {X 0,Y 428.615,Z 295.143,A -85,B 0,C 180,E1 -9832.698,E2 -9832.698} C_VEL
LIN {X 0,Y 428.697,Z 292.228,A -85,B 0,C 180,E1 -9833.169,E2 -9833.169} C_VEL
LIN {X 0,Y 429.301,Z 284.181,A -85,B 0,C 180,E1 -9834.674,E2 -9834.674} C_VEL
LIN {X 0,Y 427.318,Z 273.768,A -85,B 0,C 180,E1 -9836.823,E2 -9836.823} C_VEL
LIN {X 0,Y 425.364,Z 265.246,A -85,B 0,C 180,E1 -9838.699,E2 -9838.699} C_VEL
LIN {X 0,Y 425.263,Z 265.137,A -85,B 0,C 180,E1 -9841.926,E2 -9841.926} C_VEL
LIN {X 0,Y 425.297,Z 265.133,A -85,B 0,C 180,E1 -9845.335,E2 -9845.335} C_VEL
LIN {X 0,Y 425.29,Z 265.134,A -85,B 0,C 180,E1 -9849.042,E2 -9849.042} C_VEL
LIN {X 0,Y 425.275,Z 265.127,A -85,B 0,C 180,E1 -9852.652,E2 -9852.652} C_VEL
LIN {X 0,Y 425.257,Z 265.135,A -85,B 0,C 180,E1 -9856.044,E2 -9856.044} C_VEL
LIN {X 0,Y 425.27,Z 265.132,A -85,B 0,C 180,E1 -9858.621,E2 -9858.621} C_VEL
LIN {X 0,Y 425.31,Z 265.129,A -85,B 0,C 180,E1 -9861.103,E2 -9861.103} C_VEL
LIN {X 0,Y 425.295,Z 265.106,A -85,B 0,C 180,E1 -9864.664,E2 -9864.664} C_VEL
LIN {X 0,Y 425.268,Z 265.128,A -85,B 0,C 180,E1 -9868.073,E2 -9868.073} C_VEL
LIN {X 0,Y 425.332,Z 265.125,A -85,B 0,C 180,E1 -9871.368,E2 -9871.368} C_VEL
LIN {X 0,Y 425.289,Z 265.133,A -85,B 0,C 180,E1 -9874.554,E2 -9874.554} C_VEL
LIN {X 0,Y 425.281,Z 265.128,A -85,B 0,C 180,E1 -9877.661,E2 -9877.661} C_VEL
LIN {X 0,Y 425.355,Z 265.123,A -85,B 0,C 180,E1 -9880.704,E2 -9880.704} C_VEL
LIN {X 0,Y 425.381,Z 265.114,A -85,B 0,C 180,E1 -9883.688,E2 -9883.688} C_VEL
LIN {X 0,Y 425.404,Z 265.12,A -85,B 0,C 180,E1 -9887.598,E2 -9887.598} C_VEL
LIN {X 0,Y 425.435,Z 265.112,A -85,B 0,C 180,E1 -9891.45,E2 -9891.45} C_VEL
LIN {X 0,Y 425.546,Z 265.095,A -85,B 0,C 180,E1 -9894.313,E2 -9894.313} C_VEL
LIN {X 0,Y 425.567,Z 265.097,A -85,B 0,C 180,E1 -9898.107,E2 -9898.107} C_VEL
LIN {X 0,Y 425.695,Z 265.08,A -85,B 0,C 180,E1 -9900,E2 -9900} C_VEL
LIN {X 0,Y 425.55,Z 265.086,A -85,B 0,C 180,E1 -9902.84,E2 -9902.84} C_VEL
LIN {X 0,Y 425.523,Z 265.102,A -85,B 0,C 180,E1 -9906.642,E2 -9906.642} C_VEL
LIN {X 0,Y 425.393,Z 265.113,A -85,B 0,C 180,E1 -9909.51,E2 -9909.51} C_VEL
LIN {X 0,Y 425.387,Z 265.122,A -85,B 0,C 180,E1 -9912.904,E2 -9912.904} C_VEL
LIN {X 0,Y 425.354,Z 265.12,A -85,B 0,C 180,E1 -9916.605,E2 -9916.605} C_VEL
LIN {X 0,Y 425.321,Z 265.123,A -85,B 0,C 180,E1 -9919.636,E2 -9919.636} C_VEL
LIN {X 0,Y 425.3,Z 265.134,A -85,B 0,C 180,E1 -9923.366,E2 -9923.366} C_VEL
LIN {X 0,Y 425.342,Z 265.12,A -85,B 0,C 180,E1 -9926.845,E2 -9926.845} C_VEL
LIN {X 0,Y 425.313,Z 265.127,A -85,B 0,C 180,E1 -9929.718,E2 -9929.718} C_VEL
LIN {X 0,Y 425.277,Z 265.105,A -85,B 0,C 180,E1 -9933.049,E2 -9933.049} C_VEL
LIN {X 0,Y 425.28,Z 265.126,A -85,B 0,C 180,E1 -9935.93,E2 -9935.93} C_VEL
LIN {X 0,Y 425.306,Z 265.127,A -85,B 0,C 180,E1 -9939.046,E2 -9939.046} C_VEL
LIN {X 0,Y 425.311,Z 265.107,A -85,B 0,C 180,E1 -9941.963,E2 -9941.963} C_VEL
LIN {X 0,Y 425.286,Z 265.132,A -85,B 0,C 180,E1 -9945.283,E2 -9945.283} C_VEL
LIN {X 0,Y 425.274,Z 265.125,A -85,B 0,C 180,E1 -9948.622,E2 -9948.622} C_VEL
LIN {X 0,Y 425.31,Z 265.127,A -85,B 0,C 180,E1 -9951.104,E2 -9951.104} C_VEL
LIN {X 0,Y 425.299,Z 265.132,A -85,B 0,C 180,E1 -9954.665,E2 -9954.665} C_VEL
LIN {X 0,Y 425.264,Z 265.136,A -85,B 0,C 180,E1 -9958.074,E2 -9958.074} C_VEL
LIN {X 0,Y 425.331,Z 265.11,A -85,B 0,C 180,E1 -9961.368,E2 -9961.368} C_VEL
LIN {X 0,Y 425.396,Z 265.222,A -85,B 0,C 180,E1 -9962.538,E2 -9962.538} C_VEL
LIN {X 0,Y 427.621,Z 275.732,A -85,B 0,C 180,E1 -9964.908,E2 -9964.908} C_VEL
LIN {X 0,Y 428.976,Z 283.474,A -85,B 0,C 180,E1 -9966.558,E2 -9966.558} C_VEL
LIN {X 0,Y 428.68,Z 287.712,A -85,B 0,C 180,E1 -9967.336,E2 -9967.336} C_VEL
LIN {X 0,Y 433.643,Z 311.708,A -85,B 0,C 180,E1 -9968.058,E2 -9968.058} C_VEL
LIN {X 0,Y 432.479,Z 406.131,A -85,B 0,C 180,E1 -9969.644,E2 -9969.644} C_VEL
LIN {X 0,Y 432.044,Z 426.749,A -85,B 0,C 180,E1 -9970.026,E2 -9970.026} C_VEL
LIN {X 0,Y 431.494,Z 441.435,A -85,B 0,C 180,E1 -9970.495,E2 -9970.495} C_VEL
LIN {X 0,Y 430.869,Z 455.027,A -85,B 0,C 180,E1 -9971.126,E2 -9971.126} C_VEL
LIN {X 0,Y 430.088,Z 467.894,A -85,B 0,C 180,E1 -9971.912,E2 -9971.912} C_VEL
LIN {X 0,Y 429.196,Z 480.133,A -85,B 0,C 180,E1 -9972.858,E2 -9972.858} C_VEL
LIN {X 0,Y 428.144,Z 492.474,A -85,B 0,C 180,E1 -9974.041,E2 -9974.041} C_VEL
LIN {X 0,Y 428.05,Z 494.114,A -85,B 0,C 180,E1 -9974.225,E2 -9974.225} C_VEL
LIN {X 0,Y 427.027,Z 498.659,A -85,B 0,C 180,E1 -9974.72,E2 -9974.72} C_VEL
LIN {X 0,Y 423.578,Z 505.764,A -85,B 0,C 180,E1 -9975.525,E2 -9975.525} C_VEL
LIN {X 0,Y 420.184,Z 512.444,A -85,B 0,C 180,E1 -9976.404,E2 -9976.404} C_VEL
LIN {X 0,Y 419.259,Z 516.218,A -85,B 0,C 180,E1 -9977.009,E2 -9977.009} C_VEL
LIN {X 0,Y 418.45,Z 524.745,A -85,B 0,C 180,E1 -9978.618,E2 -9978.618} C_VEL
LIN {X 0,Y 417.88,Z 532.02,A -85,B 0,C 180,E1 -9980.318,E2 -9980.318} C_VEL
LIN {X 0,Y 417.427,Z 538.555,A -85,B 0,C 180,E1 -9982.259,E2 -9982.259} C_VEL
LIN {X 0,Y 417.301,Z 541.995,A -85,B 0,C 180,E1 -9983.542,E2 -9983.542} C_VEL
LIN {X 0,Y 417.143,Z 545.339,A -85,B 0,C 180,E1 -9985.168,E2 -9985.168} C_VEL
LIN {X 0,Y 417.032,Z 548.049,A -85,B 0,C 180,E1 -9987.102,E2 -9987.102} C_VEL
LIN {X 0,Y 416.992,Z 549.408,A -85,B 0,C 180,E1 -9989.034,E2 -9989.034} C_VEL
LIN {X 0,Y 416.992,Z 549.445,A -85,B 0,C 180,E1 -9990.966,E2 -9990.966} C_VEL
LIN {X 0,Y 417.032,Z 548.155,A -85,B 0,C 180,E1 -9992.898,E2 -9992.898} C_VEL
LIN {X 0,Y 417.144,Z 545.51,A -85,B 0,C 180,E1 -9994.832,E2 -9994.832} C_VEL
LIN {X 0,Y 417.321,Z 541.44,A -85,B 0,C 180,E1 -9996.77,E2 -9996.77} C_VEL
LIN {X 0,Y 417.638,Z 535.819,A -85,B 0,C 180,E1 -9998.711,E2 -9998.711} C_VEL
LIN {X 0,Y 418.128,Z 529.471,A -85,B 0,C 180,E1 -10000.41,E2 -10000.41} C_VEL
LIN {X 0,Y 418.773,Z 521.578,A -85,B 0,C 180,E1 -10002.109,E2 -10002.109} C_VEL
LIN {X 0,Y 419.517,Z 512.656,A -85,B 0,C 180,E1 -10003.675,E2 -10003.675} C_VEL
LIN {X 0,Y 420.325,Z 503.373,A -85,B 0,C 180,E1 -10005.02,E2 -10005.02} C_VEL
LIN {X 0,Y 421.317,Z 492.3,A -85,B 0,C 180,E1 -10006.349,E2 -10006.349} C_VEL
LIN {X 0,Y 422.316,Z 481.274,A -85,B 0,C 180,E1 -10007.43,E2 -10007.43} C_VEL
LIN {X 0,Y 423.256,Z 469.308,A -85,B 0,C 180,E1 -10008.39,E2 -10008.39} C_VEL
LIN {X 0,Y 424.101,Z 456.043,A -85,B 0,C 180,E1 -10009.232,E2 -10009.232} C_VEL
LIN {X 0,Y 424.819,Z 442.341,A -85,B 0,C 180,E1 -10009.887,E2 -10009.887} C_VEL
LIN {X 0,Y 425.449,Z 428.052,A -85,B 0,C 180,E1 -10010.36,E2 -10010.36} C_VEL
LIN {X 0,Y 425.801,Z 408.127,A -85,B 0,C 180,E1 -10010.753,E2 -10010.753} C_VEL
LIN {X 0,Y 427.15,Z 313.546,A -85,B 0,C 180,E1 -10012.359,E2 -10012.359} C_VEL
LIN {X 0,Y 421.946,Z 288.08,A -85,B 0,C 180,E1 -10013.128,E2 -10013.128} C_VEL
LIN {X 0,Y 421.949,Z 286.759,A -85,B 0,C 180,E1 -10013.302,E2 -10013.302} C_VEL
LIN {X 0,Y 421.874,Z 282.919,A -85,B 0,C 180,E1 -10014.087,E2 -10014.087} C_VEL
LIN {X 0,Y 419.234,Z 270.184,A -85,B 0,C 180,E1 -10016.912,E2 -10016.912} C_VEL
LIN {X 0,Y 418.38,Z 266.304,A -85,B 0,C 180,E1 -10017.815,E2 -10017.815} C_VEL
LIN {X 0,Y 418.295,Z 265.982,A -85,B 0,C 180,E1 -10018.062,E2 -10018.062} C_VEL
LIN {X 0,Y 418.21,Z 266.011,A -85,B 0,C 180,E1 -10021.395,E2 -10021.395} C_VEL
LIN {X 0,Y 418.264,Z 266.004,A -85,B 0,C 180,E1 -10024.58,E2 -10024.58} C_VEL
LIN {X 0,Y 418.227,Z 266.005,A -85,B 0,C 180,E1 -10027.833,E2 -10027.833} C_VEL
LIN {X 0,Y 418.221,Z 266.014,A -85,B 0,C 180,E1 -10030.947,E2 -10030.947} C_VEL
LIN {X 0,Y 418.213,Z 266.009,A -85,B 0,C 180,E1 -10033.73,E2 -10033.73} C_VEL
LIN {X 0,Y 418.205,Z 266.012,A -85,B 0,C 180,E1 -10036.448,E2 -10036.448} C_VEL
LIN {X 0,Y 418.261,Z 265.987,A -85,B 0,C 180,E1 -10039.123,E2 -10039.123} C_VEL
LIN {X 0,Y 418.233,Z 266.013,A -85,B 0,C 180,E1 -10042.164,E2 -10042.164} C_VEL
LIN {X 0,Y 418.26,Z 265.987,A -85,B 0,C 180,E1 -10045.419,E2 -10045.419} C_VEL
LIN {X 0,Y 418.21,Z 266,A -85,B 0,C 180,E1 -10048.604,E2 -10048.604} C_VEL
LIN {X 0,Y 418.288,Z 266.004,A -85,B 0,C 180,E1 -10051.936,E2 -10051.936} C_VEL
LIN {X 0,Y 418.283,Z 266.006,A -85,B 0,C 180,E1 -10055.162,E2 -10055.162} C_VEL
LIN {X 0,Y 418.226,Z 266.009,A -85,B 0,C 180,E1 -10058.303,E2 -10058.303} C_VEL
LIN {X 0,Y 418.276,Z 266.007,A -85,B 0,C 180,E1 -10061.383,E2 -10061.383} C_VEL
LIN {X 0,Y 418.294,Z 265.999,A -85,B 0,C 180,E1 -10064.406,E2 -10064.406} C_VEL
LIN {X 0,Y 418.347,Z 265.997,A -85,B 0,C 180,E1 -10067.385,E2 -10067.385} C_VEL
LIN {X 0,Y 418.334,Z 265.995,A -85,B 0,C 180,E1 -10070.328,E2 -10070.328} C_VEL
LIN {X 0,Y 418.486,Z 265.979,A -85,B 0,C 180,E1 -10073.249,E2 -10073.249} C_VEL
LIN {X 0,Y 418.334,Z 265.997,A -85,B 0,C 180,E1 -10075.181,E2 -10075.181} C_VEL
LIN {X 0,Y 418.536,Z 265.96,A -85,B 0,C 180,E1 -10078.075,E2 -10078.075} C_VEL
LIN {X 0,Y 418.665,Z 265.955,A -85,B 0,C 180,E1 -10080,E2 -10080} C_VEL
LIN {X 0,Y 418.503,Z 265.97,A -85,B 0,C 180,E1 -10082.888,E2 -10082.888} C_VEL
LIN {X 0,Y 418.485,Z 265.982,A -85,B 0,C 180,E1 -10086.751,E2 -10086.751} C_VEL
LIN {X 0,Y 418.392,Z 265.987,A -85,B 0,C 180,E1 -10088.695,E2 -10088.695} C_VEL
LIN {X 0,Y 418.307,Z 265.995,A -85,B 0,C 180,E1 -10091.631,E2 -10091.631} C_VEL
LIN {X 0,Y 418.295,Z 266.001,A -85,B 0,C 180,E1 -10094.597,E2 -10094.597} C_VEL
LIN {X 0,Y 418.28,Z 265.999,A -85,B 0,C 180,E1 -10097.604,E2 -10097.604} C_VEL
LIN {X 0,Y 418.242,Z 266.006,A -85,B 0,C 180,E1 -10100.663,E2 -10100.663} C_VEL
LIN {X 0,Y 418.28,Z 266.003,A -85,B 0,C 180,E1 -10103.782,E2 -10103.782} C_VEL
LIN {X 0,Y 418.303,Z 265.994,A -85,B 0,C 180,E1 -10107.071,E2 -10107.071} C_VEL
LIN {X 0,Y 418.256,Z 266.01,A -85,B 0,C 180,E1 -10110.271,E2 -10110.271} C_VEL
LIN {X 0,Y 418.243,Z 265.984,A -85,B 0,C 180,E1 -10113.678,E2 -10113.678} C_VEL
LIN {X 0,Y 418.24,Z 266.005,A -85,B 0,C 180,E1 -10117.224,E2 -10117.224} C_VEL
LIN {X 0,Y 418.25,Z 266.009,A -85,B 0,C 180,E1 -10119.682,E2 -10119.682} C_VEL
LIN {X 0,Y 418.225,Z 266.013,A -85,B 0,C 180,E1 -10122.322,E2 -10122.322} C_VEL
LIN {X 0,Y 418.254,Z 266.008,A -85,B 0,C 180,E1 -10125.113,E2 -10125.113} C_VEL
LIN {X 0,Y 418.289,Z 265.991,A -85,B 0,C 180,E1 -10127.774,E2 -10127.774} C_VEL
LIN {X 0,Y 418.262,Z 266.007,A -85,B 0,C 180,E1 -10131.56,E2 -10131.56} C_VEL
LIN {X 0,Y 418.256,Z 266.012,A -85,B 0,C 180,E1 -10135.16,E2 -10135.16} C_VEL
LIN {X 0,Y 418.243,Z 266.011,A -85,B 0,C 180,E1 -10137.473,E2 -10137.473} C_VEL
LIN {X 0,Y 418.3,Z 266.107,A -85,B 0,C 180,E1 -10140.943,E2 -10140.943} C_VEL
LIN {X 0,Y 420.114,Z 273.835,A -85,B 0,C 180,E1 -10142.697,E2 -10142.697} C_VEL
LIN {X 0,Y 422.415,Z 285.505,A -85,B 0,C 180,E1 -10145.16,E2 -10145.16} C_VEL
LIN {X 0,Y 421.751,Z 294.713,A -85,B 0,C 180,E1 -10146.877,E2 -10146.877} C_VEL
LIN {X 0,Y 424.266,Z 307.331,A -85,B 0,C 180,E1 -10147.281,E2 -10147.281} C_VEL
LIN {X 0,Y 427.075,Z 322.729,A -85,B 0,C 180,E1 -10147.713,E2 -10147.713} C_VEL
LIN {X 0,Y 425.549,Z 427.042,A -85,B 0,C 180,E1 -10149.487,E2 -10149.487} C_VEL
LIN {X 0,Y 425.082,Z 441.225,A -85,B 0,C 180,E1 -10149.842,E2 -10149.842} C_VEL
LIN {X 0,Y 424.471,Z 454.381,A -85,B 0,C 180,E1 -10150.348,E2 -10150.348} C_VEL
LIN {X 0,Y 423.63,Z 468.426,A -85,B 0,C 180,E1 -10151.092,E2 -10151.092} C_VEL
LIN {X 0,Y 422.738,Z 481.033,A -85,B 0,C 180,E1 -10151.963,E2 -10151.963} C_VEL
LIN {X 0,Y 421.695,Z 493.538,A -85,B 0,C 180,E1 -10153.043,E2 -10153.043} C_VEL
LIN {X 0,Y 420.715,Z 504.845,A -85,B 0,C 180,E1 -10154.25,E2 -10154.25} C_VEL
LIN {X 0,Y 419.826,Z 514.229,A -85,B 0,C 180,E1 -10155.458,E2 -10155.458} C_VEL
LIN {X 0,Y 418.996,Z 524.175,A -85,B 0,C 180,E1 -10157,E2 -10157} C_VEL
LIN {X 0,Y 418.32,Z 532.665,A -85,B 0,C 180,E1 -10158.615,E2 -10158.615} C_VEL
LIN {X 0,Y 417.733,Z 539.93,A -85,B 0,C 180,E1 -10160.315,E2 -10160.315} C_VEL
LIN {X 0,Y 417.316,Z 546.459,A -85,B 0,C 180,E1 -10162.257,E2 -10162.257} C_VEL
LIN {X 0,Y 417.122,Z 551.344,A -85,B 0,C 180,E1 -10164.198,E2 -10164.198} C_VEL
